//--------------------------------------------------------------------------------------
// Cyclic action
	IF (stStateMachine.intState=stStateMachine.intStateLastCycle) THEN
		// Simulation
		IF (SIf.stCfg.bolSimulation) THEN
			IF (((SIf.stMove.lreActPos+fbMcRelMove.Distance)<SIf.stMove.lreSWLimitPos_mm) AND (fbMcRelMove.Distance>0)AND (SIf.stMove.lreActPos<(lreActPos_old+fbMcRelMove.Distance))) THEN
				SIf.stMove.lreActPos := SIf.stMove.lreActPos + (fbMcRelMove.Velocity*udiSimPosTime_ms)/1000;
				SIf.stMove.lreActVel := fbMcRelMove.Velocity;
				SIf.stStatus.bolInPos := FALSE;
			ELSIF (((SIf.stMove.lreActPos+fbMcRelMove.Distance)>SIf.stMove.lreSWLimitNeg_mm) AND (fbMcRelMove.Distance<0)AND (SIf.stMove.lreActPos>(lreActPos_old+fbMcRelMove.Distance))) THEN
				SIf.stMove.lreActPos := SIf.stMove.lreActPos - (fbMcRelMove.Velocity*udiSimPosTime_ms)/1000;
				SIf.stMove.lreActVel := fbMcRelMove.Velocity;
				SIf.stStatus.bolInPos := FALSE;
			ELSE
				SIf.stMove.lreSetSpeed := 0;
				SIf.stStatus.bolInPos := TRUE;
			END_IF
		END_IF

		// No change action
		//MC_MoveRelative starts a relative positioning procedure based on the current set position and monitors the axis movement over the whole travel path.
		fbMcRelMove.Velocity := SIf.stMove.lreSetSpeed;
		fbMcRelMove.Deceleration := SIf.stMove.lreSetDec;
		fbMcRelMove.Acceleration := SIf.stMove.lreSetAcc;
		fbMcRelMove.Jerk := SIf.stMove.lreSetJerk;
		fbMcRelMove.Distance := SIf.stMove.lreSetPos;
		fbMcRelMove.Execute := TRUE;
		
		// State Change Condition
		IF (fbMcRelMove.Error) AND (bolfpFirstCycleDone) THEN
			SIf.stErr.dwoErrorID := fbMcRelMove.ErrorID;
			stStateMachine.intStateNext := cPOD_STA_Error;
		ELSIF (SIf.intCmd=cPOD_CMD_STOP) THEN
			stStateMachine.intStateNext := cPOD_STA_StopBusy;
		ELSIF (SIf.intCmd<>cPOD_CMD_REL_MOVE) THEN
			stStateMachine.intStateNext := cPOD_STA_QStopBusy;
		ELSIF ((SIf.stCfg.bolSimulation AND SIf.stStatus.bolInPos) OR (fbMcRelMove.Done))  AND (bolfpFirstCycleDone) THEN
			IF (SIf.intCmd=cPOD_CMD_REL_MOVE) THEN
				SIf.intCmd := cPOD_CMD_DONE;
			END_IF;
			stStateMachine.intStateNext := cPOD_STA_WaitForJob;
		END_IF
		bolfpFirstCycleDone := TRUE; //at least one call at the end of the FUB needed!
	END_IF

//--------------------------------------------------------------------------------------
// Exit action
	IF (stStateMachine.intState<>stStateMachine.intStateNext) THEN
		fbMcRelMove.Execute := FALSE;
		IF (SIf.stCfg.bolSimulation) THEN
			SIf.stMove.lreActVel := 0;
		END_IF
	END_IF
END_METHOD

{attribute 'object_name' := 'sta_StopBusy'}
METHOD PROTECTED sta_StopBusy : BOOL
// state implemetation
//--------------------------------------------------------------------------------------
// Entry action
	IF (stStateMachine.intState<>stStateMachine.intStateLastCycle) THEN
		stStateMachine.intStateLastCycle := stStateMachine.intState;
		
		bolfpFirstCycleDone := FALSE;
		
		IF (SIf.stCfg.bolSimulation) THEN
			SIf.stMove.lreActVel := 0;
		END_IF
	END_IF


//--------------------------------------------------------------------------------------
// Cyclic action
	IF (stStateMachine.intState=stStateMachine.intStateLastCycle) THEN

		//MC_Stop stops an axis with a defined braking ramp and blocks the axis for any motion commands. This behavior qualifies the block for stops under special circumstances where the axis must be prevented from further motion.
		fbMcHalt.Deceleration := SIf.stMove.lreSetDec;
		fbMcHalt.Jerk := 0; //Jerk (≥0). If the value is 0, the jerk parameterised with the last Move command is used.
		fbMcHalt.Execute := TRUE;
	
		// State Change Condition
		IF (fbMcHalt.Error) THEN
			SIf.stErr.dwoErrorID := fbMcHalt.ErrorID;
			stStateMachine.intStateNext := cPOD_STA_Error;
		ELSIF (fbMcHalt.Done) OR (SIf.stCfg.bolSimulation) THEN
			IF (SIf.intCmd=cPOD_CMD_STOP) THEN
				SIf.intCmd := cPOD_CMD_DONE;
			END_IF;
			stStateMachine.intStateNext := cPOD_STA_WaitForJob;
		ELSIF (SIf.intCmd=cPOD_CMD_CTRL_OFF) THEN
			stStateMachine.intStateNext := cPOD_STA_QStopBusy;
		END_IF
		bolfpFirstCycleDone := TRUE; //at least one call at the end of the FUB needed!
	END_IF




//--------------------------------------------------------------------------------------
// Exit action
	IF (stStateMachine.intState<>stStateMachine.intStateNext) THEN
		fbMcHalt.Execute := FALSE;
	END_IF
END_METHOD

{attribute 'object_name' := 'sta_WaitForJob'}
METHOD PROTECTED sta_WaitForJob : BOOL
// state implemetation
//--------------------------------------------------------------------------------------
// Entry action
	IF (stStateMachine.intState<>stStateMachine.intStateLastCycle) THEN
		stStateMachine.intStateLastCycle := stStateMachine.intState;
		
	END_IF


//--------------------------------------------------------------------------------------
// Cyclic action
	IF (stStateMachine.intState=stStateMachine.intStateLastCycle) THEN

		// State Change Condition
		IF (SIf.intCmd=cPOD_CMD_CTRL_OFF) THEN
			stStateMachine.intStateNext := cPOD_STA_PowerOff;
		ELSIF (SIf.intCmd=cPOD_CMD_CTRL_ON) THEN
			SIf.intCmd := cPOD_CMD_DONE;
		ELSIF (SIf.intCmd=cPOD_CMD_HOME) THEN
			stStateMachine.intStateNext := cPOD_STA_HomeBusy;
		ELSIF (SIf.intCmd=cPOD_CMD_REL_MOVE) THEN
			stStateMachine.intStateNext := cPOD_STA_RelMoveBusy;
		ELSIF (SIf.intCmd=cPOD_CMD_ABS_MOVE) THEN
			stStateMachine.intStateNext := cPOD_STA_AbsMoveBusy;
		ELSIF (SIf.intCmd=cPOD_CMD_MOD_MOVE) THEN
			stStateMachine.intStateNext := cPOD_STA_ModMoveBusy;
		ELSIF (SIf.intCmd=cPOD_CMD_POS_MOVE) THEN
			stStateMachine.intStateNext := cPOD_STA_PosMoveBusy;
		ELSIF (SIf.intCmd=cPOD_CMD_NEG_MOVE) THEN
			stStateMachine.intStateNext := cPOD_STA_NegMoveBusy;
		ELSIF (SIf.intCmd=cPOD_CMD_POS_JOG) THEN
			stStateMachine.intStateNext := cPOD_STA_PosJogBusy;
		ELSIF (SIf.intCmd=cPOD_CMD_NEG_JOG) THEN
			stStateMachine.intStateNext := cPOD_STA_NegJogBusy;
		ELSIF (SIf.intCmd=cPOD_CMD_STOP) THEN
			stStateMachine.intStateNext := cPOD_STA_StopBusy;
		ELSIF (SIf.intCmd=cPOD_CMD_EMCY_STOP_CTRL_OFF) THEN
			stStateMachine.intStateNext := cPOD_STA_QStopBusy;	
		END_IF
		
	END_IF


//--------------------------------------------------------------------------------------
// Exit action
	IF (stStateMachine.intState<>stStateMachine.intStateNext) THEN
		;
	END_IF
END_METHOD

{attribute 'object_name' := 'StateMachine'}
METHOD PROTECTED StateMachine : BOOL

// main statemachine of base controller
CASE stStateMachine.intState OF
	cPOD_STA_PowerOff: 
        THIS^.sta_PowerOff();
    cPOD_STA_PowerOnBusy: 
        THIS^.sta_PowerOnBusy();
	cPOD_STA_WaitForJob: 
        THIS^.sta_WaitForJob();
    cPOD_STA_HomeBusy: 
        THIS^.sta_HomeBusy();
	cPOD_STA_RelMoveBusy: 
        THIS^.sta_RelMoveBusy();
    cPOD_STA_AbsMoveBusy: 
        THIS^.sta_AbsMoveBusy();
	cPOD_STA_ModMoveBusy: 
        THIS^.sta_ModMoveBusy();
	cPOD_STA_PosMoveBusy: 
        THIS^.sta_PosMoveBusy();
	cPOD_STA_PosJogBusy: 
        THIS^.sta_PosJogBusy();
	cPOD_STA_NegMoveBusy: 
        THIS^.sta_NegMoveBusy();
	cPOD_STA_NegJogBusy: 
        THIS^.sta_NegJogBusy();
	cPOD_STA_QStopBusy: 
        THIS^.sta_QStopBusy();
	cPOD_STA_StopBusy: 
        THIS^.sta_StopBusy();
    cPOD_STA_Error: 
        THIS^.sta_Error();
END_CASE;
END_METHOD

{attribute 'object_name' := 'StateMachine_Service'}
METHOD PROTECTED StateMachine_Service : BOOL

IF (SIf.stCfg.bolSimulation) THEN
	SIf.stService.strValue := 'not available in simulation';
	SIf.intServiceCmd := cPOD_CMD_DONE;
ELSE

	// main statemachine of base controller
	CASE SIf.intServiceCmd OF
		cPOD_SCMD_WRITE_PARA: 
			THIS^.sJobWriteParameter();
		cPOD_SCMD_READ_PARA: 
			THIS^.sJobReadParameter();
		cPOD_SCMD_READ_PARA_NC: 
			THIS^.sJobReadParameterNC();
		cPOD_SCMD_WRITE_PARA_NC: 
			THIS^.sJobWriteParameterNC();
	ELSE
		SIf.intServiceCmd := POD_Cmd.cPOD_CMD_DONE;	
	END_CASE;
	
	// reset fb in same cycle as reset job -> done -> next job 
	IF (SIf.intServiceCmd = POD_Cmd.cPOD_CMD_DONE) THEN
		
		usiCaseScmd := 0;
		
		// reset FB calls - no cyclic calls!
		IF (fbEcCoeSdoWrite.bExecute) THEN
			fbEcCoeSdoWrite.bExecute := FALSE;
			fbEcCoeSdoWrite();
		END_IF
		IF (fbEcCoeSdoRead.bExecute) THEN
			fbEcCoeSdoRead.bExecute := FALSE;
			fbEcCoeSdoRead();
		END_IF
		IF (fbMCReadParameter.Enable) THEN
			fbMCReadParameter.Enable := FALSE;
			fbMCReadParameter(Axis := fbAxis);
		END_IF
		IF (fbMCReadBoolParameter.Enable) THEN
			fbMCReadBoolParameter.Enable := FALSE;
			fbMCReadBoolParameter(Axis := fbAxis);
		END_IF
		IF (fbMCWriteParameter.Execute) THEN
			fbMCWriteParameter.Execute := FALSE;
			fbMCWriteParameter(Axis := fbAxis);
		END_IF
		IF (fbMCWriteBoolParameter.Execute) THEN
			fbMCWriteBoolParameter.Execute := FALSE;
			fbMCWriteBoolParameter(Axis := fbAxis);
		END_IF
	END_IF
END_IF
END_METHOD

END_FUNCTION_BLOCK

// POUs/Controller/Driver/PTR [Paper Tracker]/FB_PTR
FUNCTION_BLOCK PUBLIC FB_PTR
VAR_INPUT
	In_uinBeltSpeed		: UINT;
END_VAR
VAR_OUTPUT
END_VAR
VAR
	m_udiTimeBase_us			: UDINT;		// Time base in [usec]
	m_intPaperOnBelt			: INT;			// # of Paper on the belt 
	m_intFirstPaperIdx			: INT;			// Index of the leading paper on the belt
	m_intLastPaperIdx			: INT;			// Index of the last paper on the belt
	m_arBuffer					: ARRAY[0..THIS^.cMAXBUFFERSIZE-1] OF T_PTR_STRUCT;
	m_arPositionList			: ARRAY[0..THIS^.cMAXBUFFERSIZE-1] OF T_PTR_STRUCT;
	m_intPaperEntryOffset_mm	: INT;
	m_dinBeltLength				: DINT;
	
	iIdx					: INT;
	iNdx					: INT;
	iDifference				: DINT;
END_VAR
VAR CONSTANT
	cMAXBUFFERSIZE					: INT  := 20;
	cPAPERPOSITION_TOLERANCE_mm		: UINT := 200;
END_VAR

IF m_intPaperOnBelt > 0 THEN
	iNdx := m_intFirstPaperIdx;
	
	FOR iIdx := 0 TO m_intPaperOnBelt-1 DO
		m_arBuffer[iNdx].udiTimeOnBelt_us := m_arBuffer[iNdx].udiTimeOnBelt_us + THIS^.m_udiTimeBase_us;
		m_arBuffer[iNdx].lrePositionOnBelt_mm := m_arBuffer[iNdx].lrePositionOnBelt_mm + UDINT_TO_LREAL(THIS^.m_udiTimeBase_us) * UDINT_TO_LREAL(THIS^.In_uinBeltSpeed) / 1000000.0;
				
		CASE m_arBuffer[iNdx].eStatus OF
			E_PTR_Status.EnterBusy:
				m_arBuffer[iNdx].lrePositionOnBeltAdjusted_mm := MIN(m_intPaperEntryOffset_mm, LREAL_TO_INT(m_arBuffer[iNdx].lrePositionOnBelt_mm));
				iDifference := m_intPaperEntryOffset_mm - LREAL_TO_DINT(m_arBuffer[iNdx].lrePositionOnBelt_mm);
					
				IF 	(iDifference < 0) AND (ABS(iDifference) > cPAPERPOSITION_TOLERANCE_mm) THEN
					m_arBuffer[iNdx].eStatus := E_PTR_Status.ERROR;
				END_IF
			E_PTR_Status.OnBelt:
				m_arBuffer[iNdx].lrePositionOnBeltAdjusted_mm := MIN(m_dinBeltLength, LREAL_TO_DINT(m_arBuffer[iNdx].lrePositionOnBelt_mm));
				iDifference := m_dinBeltLength - LREAL_TO_DINT(m_arBuffer[iNdx].lrePositionOnBelt_mm);

				IF 	(iDifference < 0) AND (ABS(iDifference) > cPAPERPOSITION_TOLERANCE_mm) THEN
					m_arBuffer[iNdx].eStatus :=  E_PTR_Status.ERROR;
				END_IF
			E_PTR_Status.ExitBusy:
		END_CASE
		
		m_arPositionList[iIdx] :=  m_arBuffer[iNdx];	
		iNdx := (iNdx + 1) MOD THIS^.cMAXBUFFERSIZE;
	END_FOR
ELSE
	m_arPositionList[0].eStatus := E_PTR_Status.Gone;
END_IF

PROPERTY PUBLIC BeltLength : DINT
GET
BeltLength := m_dinBeltLength;
END_GET
SET
m_dinBeltLength := BeltLength;
END_SET
END_PROPERTY

METHOD PUBLIC EnterComplete : BOOL
VAR_INPUT
END_VAR
m_arBuffer[m_intLastPaperIdx].eStatus := E_PTR_Status.OnBelt;
m_arBuffer[m_intLastPaperIdx].lrePositionOnBelt_mm := INT_TO_LREAL(m_intPaperEntryOffset_mm);
m_arBuffer[m_intLastPaperIdx].lrePositionOnBeltAdjusted_mm := INT_TO_LREAL(m_intPaperEntryOffset_mm);
END_METHOD

METHOD FB_init : BOOL
VAR_INPUT
	bInitRetains : BOOL; // if TRUE, the retain variables are initialized (warm start / cold start)
	bInCopyCode : BOOL;  // if TRUE, the instance afterwards gets moved into the copy code (online change)
END_VAR
m_udiTimeBase_us := 2000;
m_intPaperEntryOffset_mm := 0;
Reset();
END_METHOD

METHOD PUBLIC Insert : BOOL
VAR_INPUT
	uinPosition_mm			: UINT;
	udiItemId				: UDINT;
END_VAR
VAR
	iIdx					: INT;
	iNdx					: INT;
	iInsertIdx				: INT;
END_VAR
iInsertIdx := m_intFirstPaperIdx;
iNdx := m_intFirstPaperIdx;
iIdx := 0;
	
WHILE (iIdx < m_intPaperOnBelt) AND (uinPosition_mm < m_arBuffer[iNdx].lrePositionOnBelt_mm) DO
	iIdx := iIdx + 1;
	iNdx := (iNdx + 1) MOD THIS^.cMAXBUFFERSIZE;
END_WHILE
END_METHOD

PROPERTY PUBLIC PaperEntryOffset : INT
GET
PaperEntryOffset := m_intPaperEntryOffset_mm;
END_GET
SET
m_intPaperEntryOffset_mm := PaperEntryOffset;
END_SET
END_PROPERTY

PROPERTY PUBLIC PaperOnBelt : UINT
GET
PaperOnBelt := INT_TO_UINT(m_intPaperOnBelt);
END_GET
SET
END_SET
END_PROPERTY

METHOD PUBLIC Pop : T_PTR_STRUCT
// Remove a paper from the buffer
VAR_INPUT
END_VAR
Pop.eStatus := E_PTR_Status.Gone;
Pop.lrePositionOnBelt_mm := 0.0;
Pop.lrePositionOnBeltAdjusted_mm := 0.0;
Pop.udiItemId := 0;
Pop.udiTimeOnBelt_us := 0;


IF m_intPaperOnBelt > 0 THEN
	Pop := m_arBuffer[m_intFirstPaperIdx];
	m_arBuffer[m_intFirstPaperIdx].udiItemId := 0;
	m_arBuffer[m_intFirstPaperIdx].lrePositionOnBelt_mm := 0.0;
	m_arBuffer[m_intFirstPaperIdx].lrePositionOnBeltAdjusted_mm := 0.0;
	m_arBuffer[m_intFirstPaperIdx].udiTimeOnBelt_us := 0;
	m_arBuffer[m_intFirstPaperIdx].eStatus := E_PTR_Status.Gone;
	m_intPaperOnBelt := m_intPaperOnBelt - 1;

	IF m_intPaperOnBelt = 0 THEN
		m_arPositionList[0] := m_arBuffer[m_intFirstPaperIdx];
	END_IF

	m_intFirstPaperIdx := (m_intFirstPaperIdx + 1) MOD THIS^.cMAXBUFFERSIZE;
END_IF
END_METHOD

PROPERTY PUBLIC PositionList : POINTER TO T_PTR_STRUCT
GET
VAR
	iIdx			: INT;
	iNdx			: INT;
END_VAR
PositionList := ADR(m_arPositionList);
END_GET
SET
END_SET
END_PROPERTY

METHOD PUBLIC Push : BOOL
// Add (Push) a paper into the buffer
// Return an ID for the paper
VAR_INPUT
	In_udiItemId			: UDINT;
END_VAR
Push := FALSE;

IF m_intPaperOnBelt < THIS^.cMAXBUFFERSIZE THEN
	m_intLastPaperIdx := (m_intLastPaperIdx + 1) MOD THIS^.cMAXBUFFERSIZE;
	m_arBuffer[m_intLastPaperIdx].udiItemId := In_udiItemId;
	m_arBuffer[m_intLastPaperIdx].lrePositionOnBelt_mm := 0.0;
	m_arBuffer[m_intLastPaperIdx].lrePositionOnBeltAdjusted_mm := 0.0;
	m_arBuffer[m_intLastPaperIdx].udiTimeOnBelt_us := 0;
	m_arBuffer[m_intLastPaperIdx].eStatus := E_PTR_Status.EnterBusy;
	m_intPaperOnBelt := m_intPaperOnBelt + 1;
	Push := TRUE;
END_IF
END_METHOD

METHOD PUBLIC Reset : BOOL
VAR_INPUT
END_VAR
m_intFirstPaperIdx := 0;
m_intLastPaperIdx := -1;
m_intPaperOnBelt := 0;
END_METHOD

PROPERTY PUBLIC TimeBase : UDINT
GET
TimeBase := m_udiTimeBase_us;
END_GET
SET
m_udiTimeBase_us := TimeBase;
END_SET
END_PROPERTY

END_FUNCTION_BLOCK

// POUs/Controller/Driver/TCP (TCP communication driver)/FB_TCP
FUNCTION_BLOCK FB_TCP EXTENDS FB_CtrlBase
VAR
	/// Specific interface struct for public access
	SIf: T_Ctrl_SIf_TCP;
	intSendState: INT := 0;
	fbClientConnection: TC2_TCPIP.FB_ClientServerConnection;
	fbSend: TC2_TCPIP.FB_SocketSend;
	fbReceive: TC2_TCPIP.FB_SocketReceive;
	/// buffer for received messages
	fbReceiveBuffer: FB_DataSetFifo;
	/// buffer for messages to be sent
	fbSendBuffer: FB_DataSetFifo;
	stNextHead: ST_Header;
	bReceivedAck: BOOL;
	bReceivedNack: BOOL;
	iSendSize: UDINT;
	iNumSendTry: INT;
	tonSendTime: TON;
	pSendHeader: POINTER TO ST_Header;
	pByteSend: POINTER TO ARRAY[0..MAX_DATASET_SIZE] OF BYTE;
	pReceiveHead: POINTER TO ST_Header;
	pByteReceive: POINTER TO ARRAY[0..MAX_DATASET_SIZE] OF BYTE;
	naReceiveData: ARRAY[0..MAX_DATASET_SIZE] OF BYTE;
	pReceiveData: POINTER TO ARRAY[0..MAX_DATASET_SIZE] OF BYTE;
END_VAR
VAR CONSTANT
	cSendIdle: INT := 0;
	cSendBusy: INT := 1;
	cSendWait: INT := 2;
END_VAR

(*__________________________________________________________________________________________________
¦	
¦	Vistaprint Schweiz GmbH
¦	CH - 8401 Winterthur
¦
¦	www.vistaprint.ch - info@vistaprint.ch
¦___________________________________________________________________________________________________

Function desription:



History:
Version		Date			Author		Comment
---------------------------------------------------------------------------------------------------
0.00.1		21.05.2014		AVME/DSC	Start history. Based on TCP client from jetter prototyp (Sonja Segmueller)
___________________________________________________________________________________________________*)


SUPER^();

{attribute 'object_name' := 'Always'}
METHOD PROTECTED Always : BOOL
// not inherite from base !!!  special behaviour for this TCP driver
// SUPER^.Always();

// Conditions Always
IF (me.bolChangeBackToAUTO=TRUE) THEN // switch mode to automatic switch off controller
	//me.StateMachine.intStateNext := cSTA_OFFBusy;
	me.bolChangeBackToAUTO := FALSE;
END_IF

IF (CIf.SwCfg.bolExist=FALSE) THEN // hardware of controller does not exist
	me.StateMachine.intStateNext := cSTA_SINGLE_ANSWER;
ELSE
	;
END_IF

// ----------------------------------------------------------------------------------
// cyclic actions outside of statemachine
IF (me.StateMachine.intState<>cSTA_SINGLE_ANSWER) THEN
	
	// Cyclic call of the client connection
	fbClientConnection();	
END_IF
END_METHOD

{attribute 'object_name' := 'CtrlInit'}
METHOD CtrlInit : BOOL
// one time first cyclic call
// The socket is closed
SUPER^.CtrlInit();

me.StateMachine.intStateNext := TCP_CmdState.cSTA_Close;
END_METHOD

PROPERTY CtrlSIf : POINTER TO T_Ctrl_SIf_TCP
GET
CtrlSIf := ADR(SIf);
END_GET
END_PROPERTY

{attribute 'object_name' := 'CycleEndDuty'}
METHOD PROTECTED CycleEndDuty : BOOL
SUPER^.CycleEndDuty();

SendDataSequence();
END_METHOD

{attribute 'object_name' := 'CycleStartDuty'}
METHOD PROTECTED CycleStartDuty : BOOL
SUPER^.CycleStartDuty();

ReceiveDataSequence();
END_METHOD

{attribute 'object_name' := 'FB_init'}
METHOD FB_init : BOOL
VAR_INPUT
	/// if TRUE, the retain variables are initialized (warm start / cold start)
	bInitRetains: BOOL;
	/// if TRUE, the instance afterwards gets moved into the copy code (online change)
	bInCopyCode: BOOL;
END_VAR
VAR
	iIdx: UINT;
	iLength: UINT;
END_VAR
// ------------------------------------------------------------------------------------------------------------------------
// to manually change in new FUB implementation!!!
// define valid commands for this controller
iLength := SIZEOF(CIf.Job.aCmdList)/SIZEOF(CIf.Job.aCmdList[0]);
iIdx := 0;

WHILE (iIdx < iLength) AND (CIf.Job.aCmdList[iIdx].intCmd <> cCMD_INITIALIZED) DO
	iIdx := iIdx + 1; 
END_WHILE

IF (iIdx < iLength) THEN
// Add configuration of own comands	
	CIf.Job.aCmdList[iIdx].intCmd := TCP_CmdState.cCMD_Close;
	CIf.Job.aCmdList[iIdx].strName := 'CLOSE'; 
	CIf.Job.aCmdList[iIdx].bolAvailable := TRUE;
    iIdx := iIdx + 1;
		CIf.Job.aCmdList[iIdx].intCmd := TCP_CmdState.cCMD_Connect;
	CIf.Job.aCmdList[iIdx].strName := 'CONNECT'; 
	CIf.Job.aCmdList[iIdx].bolAvailable := TRUE;
    iIdx := iIdx + 1;

ELSE
	// Error if the aCmdList Array is to small
END_IF

// set name of class/typ
CIf.Info.strType := 'FB_TCP';
CIf.Info.strFullName := 'TCP Communication Driver';

// set alarm class
SIf.Alm[E_ALM_TCP.AddToReceiveBufferFailed].eAlmClass := E_AlmClass.INFO;
SIf.Alm[E_ALM_TCP.AddToReceiveBufferFailed].strText := 'addReceiveBufferFailed'; 
SIf.Alm[E_ALM_TCP.AddToSendBufferFailed].eAlmClass := E_AlmClass.INFO;
SIf.Alm[E_ALM_TCP.AddToSendBufferFailed].strText := 'addSendBufferFailed'; 
SIf.Alm[E_ALM_TCP.GetFromReceiveBufferFailed].eAlmClass := E_AlmClass.INFO;
SIf.Alm[E_ALM_TCP.GetFromReceiveBufferFailed].strText := 'getReceiveBufferFailed'; 
SIf.Alm[E_ALM_TCP.GetFromSendBufferFailed].eAlmClass := E_AlmClass.INFO;
SIf.Alm[E_ALM_TCP.GetFromSendBufferFailed].strText := 'getSendBufferFailed'; 
SIf.Alm[E_ALM_TCP.RemoveFromReceiveBufferFailed].eAlmClass := E_AlmClass.INFO;
SIf.Alm[E_ALM_TCP.RemoveFromReceiveBufferFailed].strText := 'RemoveReceiveBufferFailed'; 
SIf.Alm[E_ALM_TCP.RemoveFromSendBufferFailed].eAlmClass := E_AlmClass.INFO;
SIf.Alm[E_ALM_TCP.RemoveFromSendBufferFailed].strText := 'RemoveSendBufferFailed'; 
SIf.Alm[E_ALM_TCP.SocketConnectionLost].eAlmClass := E_AlmClass.INFO;
SIf.Alm[E_ALM_TCP.SocketConnectionLost].strText := 'SocketLost'; 
SIf.Alm[E_ALM_TCP.NotSent].eAlmClass := BASE_PLC.E_AlmClass.INFO;
SIf.Alm[E_ALM_TCP.NotSent].strText := 'NotSent';
SIf.Alm[E_ALM_TCP.NoAckReceived].eAlmClass := BASE_PLC.E_AlmClass.INFO;
SIf.Alm[E_ALM_TCP.NoAckReceived].strText := 'NoAckReceived';
SIf.Alm[E_ALM_TCP.FubErrorClientConnection].eAlmClass := BASE_PLC.E_AlmClass.INFO;
SIf.Alm[E_ALM_TCP.FubErrorClientConnection].strText := 'FUB error - client connection. Note add. info number';
SIf.Alm[E_ALM_TCP.FubErrorSendData].eAlmClass := BASE_PLC.E_AlmClass.INFO;
SIf.Alm[E_ALM_TCP.FubErrorSendData].strText := 'FUB error - send data. Note add. info number';
SIf.Alm[E_ALM_TCP.FubErrorReceiveData].eAlmClass := BASE_PLC.E_AlmClass.INFO;
SIf.Alm[E_ALM_TCP.FubErrorReceiveData].strText := 'FUB error - receive data. Note add. info number';


// *******************************************************************************
// initial values
// *******************************************************************************

// software configuration
CIf.SwCfg.bolExist := TRUE;
CIf.SwCfg.bolEnable := TRUE;
CIf.SwCfg.bolSimulation :=  FALSE;

// configuration
SIf.Cfg.bolAutoReconnectEnable  := TRUE;


// parameter
SIF.Par.strIPAdr := '192.168.2.182'; 
SIF.Par.udiPort := 7443;
SIF.Par.tTOConnection := T#10S;
SIF.Par.tTOReceive := T#5S;
SIF.Par.tTOSend := T#5S;
SIf.Par.iMaxWaitTimeAck := T#4S; // wait for Ack before declaring it not received
SIf.Par.iMaxSendTry := 5;

SIf.Cfg.bUsingAck := TRUE;

pReceiveData := ADR(naReceiveData);
pReceiveHead := pReceiveData;
END_METHOD

{attribute 'object_name' := 'getCmdState'}
METHOD PROTECTED getCmdState : STRING
VAR_INPUT
	intCmdState: INT;
	bolState: BOOL;
END_VAR
getCmdState := SUPER^.getCmdState(intCmdState:=intCmdState,bolState:=bolState); // get global/base defined cmds/states

IF (getCmdState='') THEN // global not defined get local
	// get string cmd/state string information in runtime	
	IF (bolState=FALSE) THEN
		// States's
		CASE intCmdState OF
			TCP_CmdState.cCMD_Connect: 
				getCmdState := 'cCMD_CONNECT';
			TCP_CmdState.cCMD_Close: 
				getCmdState := 'cCMD_CLOSE';

		END_CASE;
	ELSE
		// States's
		CASE intCmdState OF
			TCP_CmdState.cSTA_Close: 
				getCmdState := 'cSTA_CLOSE';
			TCP_CmdState.cSTA_CloseBusy: 
				getCmdState := 'cSTA_CLOSEBusy';
			TCP_CmdState.cSTA_Connect: 
				getCmdState := 'cSTA_CONNECT';
			TCP_CmdState.cSTA_ConnectBusy: 
				getCmdState := 'cSTA_CONNECTBusy';			
		END_CASE;
	END_IF 
END_IF
END_METHOD

{attribute 'object_name' := 'getCtrlSIf'}
METHOD getCtrlSIf : POINTER TO T_Ctrl_SIf_TCP
getCtrlSIf := ADR(SIf);
END_METHOD

{attribute 'object_name' := 'M_Pop'}
METHOD M_Pop : BOOL
VAR_OUTPUT
	naPopMsg: ARRAY[0..MAX_DATASET_SIZE] OF BYTE;
	bPop: BOOL;
END_VAR
IF fbReceiveBuffer.nCount > 0 THEN // there is something in the receive buffer
	fbReceiveBuffer.A_Remove( pHeader => pByteReceive );
	naPopMsg := pByteReceive^;
	M_Pop := 1;
	bPop := 1;
ELSE
	M_Pop := 0;
	bPop := 0;
END_IF
END_METHOD

{attribute 'object_name' := 'M_Push'}
METHOD M_Push : BOOL
VAR_INPUT
	paPushMsg: POINTER TO ARRAY[0..MAX_DATASET_SIZE] OF BYTE;
END_VAR
VAR
	pstPushMsg: POINTER TO ST_Header;
END_VAR
// send if desired
pstPushMsg := paPushMsg;
	
fbSendBuffer.A_Add(in := paPushMsg, iAddSize := UDINT_TO_INT(pstPushMsg^.udiMsgSize + SIZEOF(ST_HEADER)) , bOk=>M_Push );

IF NOT ( M_Push ) THEN 
	pfbAlarmCtrl^.setAlarm(CIf.Info.intCtrlId,E_ALM_TCP.AddToSendBufferFailed,0,ADR(SIf.Alm),E_AlmState.RST,CIf.Job.eMe_ActivAlmClass);
	me.StateMachine.intStateNext := BASE_PLC.cSTA_ERROR;
END_IF
END_METHOD

{attribute 'object_name' := 'ReceiveDataSequence'}
METHOD PROTECTED ReceiveDataSequence : BOOL
VAR
	bSuccess: BOOL;
	nLoad: UDINT;
	stACK: ST_Header;
END_VAR
// receive data if connected
IF (fbClientConnection.eState = TC2_TCPIP.E_SocketConnectionState.eSOCKET_CONNECTED) THEN
	IF fbReceive.bBusy THEN	
		fbReceive.bExecute := FALSE;
		fbReceive.sSrvNetId := '';
		fbReceive();
		
		IF NOT (fbReceive.bBusy) THEN
			// Receive is finished => see what we got
				
			// First Check about FUB error	
			IF (fbReceive.bError = TRUE) THEN
				IF NOT (SIf.Cur.bolFubErrorActive) THEN
					SIf.Cur.bolFubErrorActive:= TRUE;																				
					pfbAlarmCtrl^.setAlarm(CIf.Info.intCtrlId,E_ALM_TCP.FubErrorReceiveData, UDINT_TO_DINT(fbReceive.nErrId),ADR(SIf.Alm),E_AlmState.RST,CIf.Job.eMe_ActivAlmClass);																						
					// Try to close the socket. Needs reconnect for socket after an error!	
					me.StateMachine.intStateNext := TCP_CmdState.cSTA_CloseBusy;					
				END_IF	
				
			// No error			
			ELSE
				// Check received data
				CASE pReceiveHead^.uinMsgId  OF
					// ACK
					// **************************
					999: 
						bReceivedAck := 1;
					
					// NACK
					// **************************
					998: 
						bReceivedNack := 1;
						
					// Valid message IDs
					// **************************
					2, 3, 4, 5, 6, 7: 
					
						fbReceiveBuffer.A_Add(in := ADR(naReceiveData), iAddSize:= UDINT_TO_INT(SIZEOF(ST_Header) + pReceiveHead^.udiMsgSize), bOk=>bSuccess , nLoad => nLoad );
						IF NOT ( bSuccess ) THEN 
							pfbAlarmCtrl^.setAlarm(CIf.Info.intCtrlId,E_ALM_TCP.AddToReceiveBufferFailed,0,ADR(SIf.Alm),E_AlmState.RST,CIf.Job.eMe_ActivAlmClass);
							me.StateMachine.intStateNext := BASE_PLC.cSTA_ERROR;
							me.StateMachine.intState := BASE_PLC.cSTA_ERROR;
						END_IF
								
					// nothing has been received	
					// **************************
					0: 
					
				ELSE
					// send NACK Command
					IF(SIf.Cfg.bUsingAck) THEN
						stACK.uinMsgId := 998;
						fbSendBuffer.A_Add(in := ADR(stACK), bOk=>bSuccess , nLoad => nLoad, iAddSize:= SIZEOF(stACK.uinMsgId) );
						IF NOT (bSuccess) THEN 
							pfbAlarmCtrl^.setAlarm(CIf.Info.intCtrlId,E_ALM_TCP.AddToSendBufferFailed,0,ADR(SIf.Alm),E_AlmState.RST,CIf.Job.eMe_ActivAlmClass);
							me.StateMachine.intStateNext := BASE_PLC.cSTA_ERROR;
							me.StateMachine.intState := BASE_PLC.cSTA_ERROR;
						END_IF
					END_IF
				
				END_CASE
				// empty the receive data
				pReceiveHead^.uinMsgId := 0;			
			END_IF	
			
		END_IF
		
	// Trigger the next data receive 
	ELSE
		fbReceive(bExecute := FALSE); // Needs new trigger!
		fbReceive.sSrvNetId := '';
		fbReceive.hSocket := fbClientConnection.hSocket;
		fbReceive.cbLen := SIZEOF(naReceiveData);
		fbReceive.pDest := ADR(naReceiveData);
		fbReceive.tTimeout := SIf.Par.tTOReceive;
		fbReceive.bExecute := TRUE;
		fbReceive();
	END_IF
END_IF 
fbReceive();
END_METHOD

{attribute 'object_name' := 'SendDataSequence'}
METHOD PROTECTED SendDataSequence : BOOL
VAR
	intI: INT;
END_VAR
// Handle Send Data
CASE intSendState OF
	cSendIdle: 
		IF fbSendBuffer.nCount > 0 AND NOT (fbSend.bBusy) AND (fbClientConnection.eState = TC2_TCPIP.E_SocketConnectionState.eSOCKET_CONNECTED) THEN // there is something in the buffer that needs to be sent
			intSendState := cSendBusy;
			
			// Remove data from buffer. Get next package.
			fbSendBuffer.A_Get(pHeader => pSendHeader);
			pByteSend := pSendHeader;
			stNextHead := pSendHeader^;
			
			IF (stNextHead.uinMsgId = 999) OR (stNextHead.uinMsgId = 998 ) THEN // ack or nack
				iSendSize := SIZEOF(stNextHead.uinMsgId);
			ELSE
				iSendSize := stNextHead.udiMsgSize + SIZEOF(ST_Header);
			END_IF
			
			// send Command
			fbSend(bExecute := FALSE, sSrvNetId := ''); 
			fbSend.sSrvNetId := ''; // SIf.Par.strIPAdr;
			fbSend.hSocket := fbClientConnection.hSocket;
			fbSend.cbLen := iSendSize;
			fbSend.pSrc := pByteSend;
			fbSend.bExecute := TRUE;
			fbSend.tTimeout := SIf.Par.tTOSend;
			fbSend(); 
		ELSE
			fbSend.bExecute := FALSE;
			fbSend.sSrvNetId := '';
			fbSend();
		END_IF	
		// *)
	cSendBusy:
		IF NOT (fbSend.bBusy) THEN // sending done
			
			// First Check about FUB error	
			IF (fbSend.bError = TRUE) THEN
				IF NOT (SIf.Cur.bolFubErrorActive) THEN
					SIf.Cur.bolFubErrorActive:= TRUE;																				
					pfbAlarmCtrl^.setAlarm(CIf.Info.intCtrlId,E_ALM_TCP.FubErrorSendData, UDINT_TO_DINT(fbSend.nErrId),ADR(SIf.Alm),E_AlmState.RST,CIf.Job.eMe_ActivAlmClass);																						
					// Try to close the socket. Needs reconnect for socket after an error!	
					me.StateMachine.intStateNext := TCP_CmdState.cSTA_CloseBusy;					
				END_IF	
			// no error			
			ELSE
				IF (stNextHead.uinMsgId > 997) OR (NOT (SIf.Cfg.bUsingAck)) THEN // the sent was ack or nack
					fbSendBuffer.A_Remove();
					intSendState := cSendIdle;
				ELSE // wair for ack
					intSendState := cSendWait;
					tonSendTime(IN := 0);
					tonSendTime.PT := SIf.Par.iMaxWaitTimeAck;
					tonSendTime(IN := 1);
				END_IF	
			END_IF
			
		END_IF
		
		fbSend.bExecute := FALSE;
		fbSend.sSrvNetId := '';
		fbSend(); // *)
		
	cSendWait:
		fbSend.bExecute := FALSE;
		fbSend.sSrvNetId := '';
		fbSend();
		tonSendTime(IN := 1);
		// Wait for the ACK
		IF bReceivedAck THEN
			fbSendBuffer.A_Remove();
			bReceivedAck := 0;
			iNumSendTry := 0; // reset for next send
			intSendState := cSendIdle;
			
		ELSIF (tonSendTime.Q) OR (bReceivedNack) THEN // timeout
			
			iNumSendTry := iNumSendTry +1;
			IF iNumSendTry >= SIf.Par.iMaxSendTry THEN
				// the signal has not been acknoledged too many times => error
				pfbAlarmCtrl^.setAlarm(CIf.Info.intCtrlId,E_ALM_TCP.NoAckReceived,0,ADR(SIf.Alm),E_AlmState.RST,CIf.Job.eMe_ActivAlmClass);
				me.StateMachine.intStateNext := BASE_PLC.cSTA_ERROR;
			ELSE // retry sending
				fbSend.bExecute := TRUE;
				fbSend(); 
				intSendState := cSendBusy;
			END_IF
			
		END_IF
END_CASE // *)
fbSend();
END_METHOD

{attribute 'object_name' := 'sta_CLOSE'}
METHOD sta_CLOSE : BOOL
// state implemetation
// --------------------------------------------------------------------------------------
// Entry action
	IF (me.StateMachine.intState<>me.StateMachine.intStateLastCycle) THEN
		me.StateMachine.intStateLastCycle := me.StateMachine.intState;
		;
		
	END_IF

// --------------------------------------------------------------------------------------
// Cyclic action
	IF (me.StateMachine.intState=me.StateMachine.intStateLastCycle) THEN
		CASE me.intCmd OF
			TCP_CmdState.cCMD_Connect:
				me.StateMachine.intStateNext := TCP_CmdState.cSTA_ConnectBusy;
		END_CASE
	END_IF

// --------------------------------------------------------------------------------------
// Exit action
	IF (me.StateMachine.intState<>me.StateMachine.intStateNext) THEN
		;
	END_IF
END_METHOD

{attribute 'object_name' := 'sta_CLOSEBusy'}
METHOD sta_CLOSEBusy : BOOL
// state implemetation
// --------------------------------------------------------------------------------------
// Entry action
	IF (me.StateMachine.intState<>me.StateMachine.intStateLastCycle) THEN
		me.StateMachine.intStateLastCycle := me.StateMachine.intState;
		
		// Reset Tx state
		intSendState:= cSendIdle;
		fbSend.bExecute:= FALSE;
		fbReceive.bExecute:= FALSE;
		iNumSendTry := 0;
		
		// Close socket
		fbClientConnection.bEnable:= FALSE;
		
		IF me.intCmd = TCP_CmdState.cCMD_Close THEN
			// clear both buffers
			fbSendBuffer.A_Reset();
			fbReceiveBuffer.A_Reset();
		END_IF
	END_IF

// --------------------------------------------------------------------------------------
// Cyclic action
	IF (me.StateMachine.intState=me.StateMachine.intStateLastCycle) THEN
		
		// Check about FUB error	
		IF (fbClientConnection.bError = TRUE) OR (fbClientConnection.nErrId <> 0) THEN
			SIf.Cur.bolFubErrorActive:= TRUE;																					
			pfbAlarmCtrl^.setAlarm(CIf.Info.intCtrlId,E_ALM_TCP.FubErrorClientConnection, UDINT_TO_DINT(fbClientConnection.nErrId),ADR(SIf.Alm),E_AlmState.RST,CIf.Job.eMe_ActivAlmClass);																			
			me.StateMachine.intStateNext := BASE_PLC.cSTA_ERROR;	
		END_IF
					
		// Wait until socket is closed	
		IF (fbClientConnection.eState = TC2_TCPIP.E_SocketConnectionState.eSOCKET_DISCONNECTED) THEN 	
			IF me.intCmd = TCP_CmdState.cCMD_Close THEN
				me.StateMachine.intStateNext := TCP_CmdState.cSTA_Close;
			ELSE
				me.StateMachine.intStateNext := TCP_CmdState.cSTA_ConnectBusy;
			END_IF

		ELSIF (SIf.Cur.bolFubErrorActive) THEN
			me.StateMachine.intStateNext := BASE_PLC.cSTA_ERROR;	
		END_IF
		
	END_IF
	
// --------------------------------------------------------------------------------------
// Exit action
	IF (me.StateMachine.intState<>me.StateMachine.intStateNext) THEN
		;
	END_IF
END_METHOD

{attribute 'object_name' := 'sta_CONNECT'}
METHOD sta_CONNECT : BOOL
// state implemetation
// --------------------------------------------------------------------------------------
// Entry action
	IF (me.StateMachine.intState<>me.StateMachine.intStateLastCycle) THEN
		me.StateMachine.intStateLastCycle := me.StateMachine.intState;

		pfbAlarmCtrl^.setAlarm(CIf.Info.intCtrlId,E_ALM_TCP.SocketConnectionLost,0,ADR(SIf.Alm),E_AlmState.CLR,CIf.Job.eMe_ActivAlmClass);
	END_IF

// --------------------------------------------------------------------------------------
// Cyclic action
	IF (me.StateMachine.intState=me.StateMachine.intStateLastCycle) THEN
		// check if connection has been lost
		IF (fbClientConnection.eState <> TC2_TCPIP.E_SocketConnectionState.eSOCKET_CONNECTED) THEN 
			pfbAlarmCtrl^.setAlarm(CIf.Info.intCtrlId,E_ALM_TCP.SocketConnectionLost,0,ADR(SIf.Alm),E_AlmState.RST,CIf.Job.eMe_ActivAlmClass);
			
			IF SIf.Cfg.bolAutoReconnectEnable THEN
				me.StateMachine.intStateNext := TCP_CmdState.cSTA_CloseBusy;
			ELSE	
				me.StateMachine.intStateNext := BASE_PLC.cSTA_ERROR;
			END_IF
		END_IF
		
		CASE me.intCmd OF
			TCP_CmdState.cCMD_Close:
				me.StateMachine.intStateNext := TCP_CmdState.cSTA_CloseBusy;
			TCP_CmdState.cCMD_Connect:
				me.StateMachine.intStateNext := TCP_CmdState.cSTA_CloseBusy;
		END_CASE
	END_IF

// --------------------------------------------------------------------------------------
// Exit action
	IF (me.StateMachine.intState<>me.StateMachine.intStateNext) THEN
		;
	END_IF
END_METHOD

{attribute 'object_name' := 'sta_CONNECTBusy'}
METHOD sta_CONNECTBusy : BOOL
// state implemetation
// --------------------------------------------------------------------------------------
// Entry action
	IF (me.StateMachine.intState<>me.StateMachine.intStateLastCycle) THEN
		me.StateMachine.intStateLastCycle := me.StateMachine.intState;
		
		// Initialize and connect socket
		fbClientConnection.nMode := 0; 	// not used
		fbClientConnection.sRemoteHost := SIf.Par.strIPAdr;
		fbClientConnection.nRemotePort := SIf.Par.udiPort;
		fbClientConnection.tReconnect := SIF.Par.tTOConnection;
		fbClientConnection.bEnable:= TRUE;
	
		// clear both buffers
		fbSendBuffer.A_Reset();
		fbReceiveBuffer.A_Reset();
		
		// reset all nessecary parameters
		bReceivedAck := 0;
		bReceivedNack := 0;
		intSendState := 0;
	END_IF


// --------------------------------------------------------------------------------------
// Cyclic action
	IF (me.StateMachine.intState=me.StateMachine.intStateLastCycle) THEN
		
		// Check about FUB error	
		IF (fbClientConnection.bError = TRUE) OR (fbClientConnection.nErrId <> 0) THEN		
			SIf.Cur.bolFubErrorActive:= TRUE;																			
			pfbAlarmCtrl^.setAlarm(CIf.Info.intCtrlId,E_ALM_TCP.FubErrorClientConnection, UDINT_TO_DINT(fbClientConnection.nErrId),ADR(SIf.Alm),E_AlmState.RST,CIf.Job.eMe_ActivAlmClass);																			
			me.StateMachine.intStateNext := BASE_PLC.cSTA_ERROR;	
		END_IF
				
		// Wait for socket handle ID and connection state
		IF (fbClientConnection.hSocket.handle <> 0) AND (fbClientConnection.eState = TC2_TCPIP.E_SocketConnectionState.eSOCKET_CONNECTED) THEN 	
			me.StateMachine.intStateNext := TCP_CmdState.cSTA_Connect;
		END_IF
		
	END_IF

// --------------------------------------------------------------------------------------
// Exit action
	IF (me.StateMachine.intState<>me.StateMachine.intStateNext) THEN
		;
	END_IF
END_METHOD

{attribute 'object_name' := 'sta_ERROR'}
METHOD PROTECTED sta_ERROR : BOOL
// state implemetation
// --------------------------------------------------------------------------------------
// Entry action
	IF (me.StateMachine.intState<>me.StateMachine.intStateLastCycle) THEN
		me.StateMachine.intStateHistory := me.StateMachine.intStateLastCycle; // -> possibillity to go back to state before error
		me.StateMachine.intStateLastCycle := me.StateMachine.intState;
		
		// Clear pending commands
		CIf.Job.intACmd:= Base_PLC.cCMD_DONE;
		CIf.Job.intMCmd:= Base_PLC.cCMD_DONE;
			
		iNumSendTry := 0;
				
		// clear both buffers
		fbSendBuffer.A_Reset();
		fbReceiveBuffer.A_Reset();
		// Reset Tx state
		intSendState:= cSendIdle;
	END_IF
	

// --------------------------------------------------------------------------------------
// Cyclic action
	IF (me.StateMachine.intState=me.StateMachine.intStateLastCycle) THEN
		
		// State Change Condition
		IF (CIf.Job.bolAlmReset = TRUE) THEN
			SIf.Cur.bolFubErrorActive:= FALSE;
			me.StateMachine.intStateNext := cSTA_ERRORQuit;
		END_IF
	END_IF

// --------------------------------------------------------------------------------------
// Exit action
	IF (me.StateMachine.intState<>me.StateMachine.intStateNext) THEN
		;
	END_IF
END_METHOD

{attribute 'object_name' := 'sta_ERRORQuit'}
METHOD PROTECTED sta_ERRORQuit : BOOL
// state implemetation
// --------------------------------------------------------------------------------------
// Entry action
	IF (me.StateMachine.intState<>me.StateMachine.intStateLastCycle) THEN
		me.StateMachine.intStateLastCycle := me.StateMachine.intState;
		;
	END_IF

// -------------------------------------------------------------------------------------
// Cyclic action
	IF (me.StateMachine.intState=me.StateMachine.intStateLastCycle) THEN
		
		IF (CIf.Job.bolAlmReset = TRUE) THEN
			CIf.Job.eMe_ActivAlmClass := E_AlmClass.NONE; // reset feedback channel for parent
			CIf.Job.bolAlmReset := FALSE;
		END_IF
		
		// State Change Condition
		IF (CIf.Job.bolAlmReset = FALSE) THEN
			// Needs reconnect for socket after an error!	
			me.StateMachine.intStateNext := TCP_CmdState.cSTA_CloseBusy;
		END_IF
	END_IF

// --------------------------------------------------------------------------------------
// Exit action
	IF (me.StateMachine.intState<>me.StateMachine.intStateNext) THEN
		;
	END_IF
END_METHOD

{attribute 'object_name' := 'StateMachine'}
METHOD PROTECTED StateMachine : BOOL
SUPER^.StateMachine();

// main statemachine of base controller
CASE me.StateMachine.intState OF
	TCP_CmdState.cSTA_Close:
		THIS^.sta_CLOSE();
    TCP_CmdState.cSTA_ConnectBusy:
		THIS^.sta_CONNECTBusy();
	TCP_CmdState.cSTA_Connect:
		THIS^.sta_CONNECT();
	TCP_CmdState.cSTA_CloseBusy:
		THIS^.sta_CLOSEBusy();
END_CASE;
END_METHOD

END_FUNCTION_BLOCK

// POUs/Controller/Utility/FiFo/FB_DataSetFifo
FUNCTION_BLOCK FB_DataSetFifo
VAR_INPUT
	bOverwrite: BOOL;
	in: POINTER TO BYTE;
	iAddSize: INT;
END_VAR
VAR_OUTPUT
	bOk: BOOL;
	nCount: UDINT;
	nLoad: UDINT;
	out: ARRAY[0..MAX_DATASET_SIZE] OF BYTE;
	pHeader: POINTER TO ST_Header;
END_VAR
VAR
	/// Buffer memory used by FB_MemRingBuffer function block 
	arrBuffer: ARRAY[0..MAX_BUFFER_SIZE] OF BYTE;
	fbBuffer: FB_MemRingBuffer;
	intLoopRemove: INT;
	intLoopReset: INT;
END_VAR
VAR CONSTANT
	MAX_BUFFER_SIZE: UDINT := 1000;
END_VAR

;

ACTION A_Add:
fbBuffer.A_AddTail( pWrite:= in,
					cbWrite:= INT_TO_UDINT(iAddSize),
					pBuffer:= ADR( arrBuffer ),
					cbBuffer:= SIZEOF( arrBuffer ),
					bOk=> bOk,
					nCount => nCount );

IF NOT bOk THEN (* overflow ? *)
	IF bOverwrite THEN
		fbBuffer.A_RemoveHead(); (* remove one oldest entry *)
		fbBuffer.A_AddTail( bOk => bOk, nCount => nCount );
	END_IF
END_IF

nLoad := (fbBuffer.cbSize * 100) / MAX_BUFFER_SIZE;
END_ACTION

ACTION A_Get:
fbBuffer.A_GetHead( pRead:= ADR( out ),
					cbRead:= SIZEOF( out ),
					pBuffer:= ADR( arrBuffer ),
					cbBuffer:= SIZEOF( arrBuffer ),
					bOk=> bOk,
					nCount => nCount );

pHeader := ADR(out);					
					
nLoad := (fbBuffer.cbSize * 100) / MAX_BUFFER_SIZE;
END_ACTION

ACTION A_Remove:
// Clean up package buffer
FOR intLoopRemove:=0 TO SIZEOF(out)-1 DO
	out[intLoopRemove]:= 0;
END_FOR

// Remove data from buffer. Get next package.
fbBuffer.A_RemoveHead( 	pRead:= ADR(out),
						cbRead:= SIZEOF(out),
						pBuffer:= ADR(arrBuffer),
						cbBuffer:= SIZEOF(arrBuffer),
						bOk=> bOk,
						nCount => nCount );
// Return						
pHeader := ADR(out);

nLoad := (fbBuffer.cbSize * 100) / MAX_BUFFER_SIZE;
END_ACTION

ACTION A_Reset:
// MEMSET not working!
//MEMSET( ADR( arrBuffer ), 0, SIZEOF( arrBuffer ) ); (* reset (optional) internal buffer *)
FOR intLoopReset:=0 TO SIZEOF(arrBuffer)-1 DO
	arrBuffer[intLoopReset]:= 0;
END_FOR

fbBuffer.A_Reset( 	bOk=> bOk,
					nCount => nCount );

nLoad := (fbBuffer.cbSize * 100) / MAX_BUFFER_SIZE;
END_ACTION

END_FUNCTION_BLOCK

// POUs/Controller/Lvl0/GRR (Granulate Remote)/helper/cycle_Grr
FUNCTION cycle_Grr : BOOL
VAR_INPUT
	pGrr: POINTER TO T_GRR;
END_VAR

pGrr^.ctrl.fbGrr.In_bolAutoMode				:= pGrr^.io.In_bolAutoMode;
pGrr^.ctrl.fbGrr.In_bolEoffOrFuseOk			:= pGrr^.io.In_bolEoffOrFuseOk;
pGrr^.ctrl.fbGrr.In_bolMainPressureError	:= pGrr^.io.In_bolMainPressureError;
pGrr^.ctrl.fbGrr.In_bolPowderLowWarning		:= pGrr^.io.In_bolPowderLowWarning;
pGrr^.ctrl.fbGrr.In_bolSystemOk				:= pGrr^.io.In_bolSystemOk;
pGrr^.ctrl.fbGrr.In_intState				:= pGrr^.io.In_intState;
pGrr^.ctrl.fbGrr.In_bolToggleBitGrn			:= pGrr^.io.In_bolToggleBitGrn;
pGrr^.ctrl.fbGrr.In_intMainPressure			:= pGrr^.io.In_intMainPressure;
pGrr^.ctrl.fbGrr();
pGrr^.io.Out_intCommand						:= pGrr^.ctrl.fbGrr.Out_intCommand;
pGrr^.io.Out_intConveyorBelt				:= pGrr^.ctrl.fbGrr.Out_intConveyorBelt;
pGrr^.io.Out_intConveyorVibrator			:= pGrr^.ctrl.fbGrr.Out_intConveyorVibrator;
pGrr^.io.Out_intPowderVibrator				:= pGrr^.ctrl.fbGrr.Out_intPowderVibrator;
pGrr^.io.Out_uinFilterClearingCycleTime_min	:= pGrr^.ctrl.fbGrr.Out_uinFilterClearingCycleTime_min;
pGrr^.io.Out_bolToggleBitGrr				:= pGrr^.ctrl.fbGrr.Out_bolToggleBitGrr;
pGrr^.io.Out_intAnalogValue					:= pGrr^.ctrl.fbGrr.Out_intAnalogValue;

END_FUNCTION

// POUs/Controller/Lvl0/GRR (Granulate Remote)/helper/init_Grr
FUNCTION init_Grr : BOOL
VAR_INPUT
	pGrr			: POINTER TO T_GRR;
	/// instance array of all controller instances
	pCtrlInst		: POINTER TO fb_CtrlBase;
	/// common interface array of all controllers (main use for PLC)
	pCtrlCIf		: POINTER TO T_Ctrl_CIf;
END_VAR

pGrr^.ctrl.fbGrr.iniAllCtrlArrays(pCtrlInst,pCtrlCIf,pGrr^.id.Grr);

END_FUNCTION

// POUs/Controller/Lvl0/GRR (Granulate Remote)/FB_GRR
FUNCTION_BLOCK FB_GRR EXTENDS FB_CtrlBase
VAR_INPUT
	In_bolSystemOk: BOOL;
	In_bolMainPressureError: BOOL;
	In_bolEoffOrFuseOk: BOOL;
	In_bolPowderLowWarning: BOOL;
	In_bolAutoMode: BOOL;
	In_intState: INT;
	In_bolToggleBitGrn: BOOL;
	In_intMainPressure: INT;
END_VAR
VAR_OUTPUT
	Out_intCommand: INT;
	Out_intConveyorBelt: INT;
	Out_intPowderVibrator: INT;
	Out_intConveyorVibrator: INT;
	Out_uinFilterClearingCycleTime_min: UINT;
	Out_bolToggleBitGrr: BOOL;
	Out_intAnalogValue: INT;
END_VAR
VAR
	/// Specific interface struct for public access
	SIf: T_Ctrl_SIf_Grr;
	
	udiToggleBitGrrTimer_ms		: UDINT;
	udiToggleBitGrnTimer_ms		: UDINT;
	bToggleBitGrnOld			: BOOL;
	bToggleBitOK				: BOOL;
END_VAR

(*__________________________________________________________________________________________________
¦	
¦	Vistaprint Schweiz GmbH
¦	CH - 8401 Winterthur
¦
¦	www.vistaprint.ch - info@vistaprint.ch
¦___________________________________________________________________________________________________

Function desription:

History:
Version		Date			Author		Comment
---------------------------------------------------------------------------------------------------
0.00.1		05.11.2014		BB			Start history
0.00.2		06.02.2015		BB			changed name from GRN to GRR
___________________________________________________________________________________________________*)

SUPER^();

{attribute 'object_name' := 'Always'}
METHOD PROTECTED Always : BOOL
SUPER^.Always();

// ----------------------------------------------------------------------------------
// cyclic actions outside of statemachine
IF (me.StateMachine.intState <> cSTA_SINGLE_ANSWER) THEN
	
	// Toggle Bit Grr
	udiToggleBitGrrTimer_ms := udiToggleBitGrrTimer_ms + me.FUBInfo.udiSample_ms;
	IF (udiToggleBitGrrTimer_ms > 200) THEN
		SIf.Out.bolToggleBitGrr.intern := NOT SIf.Out.bolToggleBitGrr.intern;
		udiToggleBitGrrTimer_ms := 0;
	END_IF
	
	// check Toggle Bit Grn
	udiToggleBitGrnTimer_ms := udiToggleBitGrnTimer_ms + me.FUBInfo.udiSample_ms;
	IF (SIf.In.bolToggleBitGrn.intern <> bToggleBitGrnOld) THEN
		bToggleBitGrnOld := SIf.In.bolToggleBitGrn.intern;
		udiToggleBitGrnTimer_ms := 0;
	END_IF
	bToggleBitOK := FALSE;
	IF (udiToggleBitGrnTimer_ms < 1000) THEN
		bToggleBitOK := TRUE;
	END_IF
	
	IF NOT (bToggleBitOK) AND (me.StateMachine.intState <> cSTA_ERROR) AND (me.StateMachine.intState <> cSTA_ERRORQuit) THEN
		pfbAlarmCtrl^.setAlarm(CIf.Info.intCtrlId,E_ALM_GRR.LostConnection,0,ADR(SIf.Alm),E_AlmState.RST,CIf.Job.eMe_ActivAlmClass);
		me.StateMachine.intStateNext := Base_CmdState.cSTA_ERROR;
	END_IF
	
	IF NOT SIf.In.bolAutoMode.intern AND bToggleBitOK THEN
		IF (SIf.Cfg.bolManualModeAllowed) THEN
			pfbAlarmCtrl^.setAlarm(CIf.Info.intCtrlId,E_ALM_GRR.ManualModeWarning,0,ADR(SIf.Alm),E_AlmState.SET,CIf.Job.eMe_ActivAlmClass);
			pfbAlarmCtrl^.setAlarm(CIf.Info.intCtrlId,E_ALM_GRR.ManualModeError,0,ADR(SIf.Alm),E_AlmState.CLR,CIf.Job.eMe_ActivAlmClass);
		ELSIF (me.StateMachine.intState <> cSTA_ERROR) AND (me.StateMachine.intState <> cSTA_ERRORQuit) THEN
			pfbAlarmCtrl^.setAlarm(CIf.Info.intCtrlId,E_ALM_GRR.ManualModeError,0,ADR(SIf.Alm),E_AlmState.RST,CIf.Job.eMe_ActivAlmClass);
			pfbAlarmCtrl^.setAlarm(CIf.Info.intCtrlId,E_ALM_GRR.ManualModeWarning,0,ADR(SIf.Alm),E_AlmState.CLR,CIf.Job.eMe_ActivAlmClass);
			me.StateMachine.intStateNext := Base_CmdState.cSTA_ERROR;
		END_IF
	ELSE
		pfbAlarmCtrl^.setAlarm(CIf.Info.intCtrlId,E_ALM_GRR.ManualModeWarning,0,ADR(SIf.Alm),E_AlmState.CLR,CIf.Job.eMe_ActivAlmClass);
	END_IF
	
	IF SIf.In.bolPowderLowWarning.intern AND bToggleBitOK THEN
		pfbAlarmCtrl^.setAlarm(CIf.Info.intCtrlId,E_ALM_GRR.LowPowderWarning,0,ADR(SIf.Alm),E_AlmState.SET,CIf.Job.eMe_ActivAlmClass);
	ELSE
		pfbAlarmCtrl^.setAlarm(CIf.Info.intCtrlId,E_ALM_GRR.LowPowderWarning,0,ADR(SIf.Alm),E_AlmState.CLR,CIf.Job.eMe_ActivAlmClass);
	END_IF
	
	// reasons are either PressureError or SystemError (EOFF/Fuse/Motor)
	IF NOT SIf.In.bolSystemOk.intern AND bToggleBitOK THEN
		IF SIf.In.bolMainPressureError.intern THEN
			pfbAlarmCtrl^.setAlarm(CIf.Info.intCtrlId,E_ALM_GRR.PressureError,0,ADR(SIf.Alm),E_AlmState.RST,CIf.Job.eMe_ActivAlmClass);
			me.StateMachine.intStateNext := Base_CmdState.cSTA_OFFBusy;
		ELSE
			pfbAlarmCtrl^.setAlarm(CIf.Info.intCtrlId,E_ALM_GRR.SystemError,0,ADR(SIf.Alm),E_AlmState.RST,CIf.Job.eMe_ActivAlmClass);
			me.StateMachine.intStateNext := Base_CmdState.cSTA_OFFBusy;
		END_IF
	END_IF
	
	// Check Parameters
	// Conveyor Belt
	IF (SIf.Par.rConveyorBelt_Hz>SIf.Cfg.rMaxFreq_Hz) THEN
		SIf.Par.rConveyorBelt_Hz := SIf.Cfg.rMaxFreq_Hz;
	ELSIF (SIf.Par.rConveyorBelt_Hz<0) THEN
		SIf.Par.rConveyorBelt_Hz := 0;
	END_IF
	// Conveyor Vibrator
	IF (SIf.Par.rConveyorVibrator_Hz>SIf.Cfg.rMaxFreq_Hz) THEN
		SIf.Par.rConveyorVibrator_Hz := SIf.Cfg.rMaxFreq_Hz;
	ELSIF (SIf.Par.rConveyorVibrator_Hz<0) THEN
		SIf.Par.rConveyorVibrator_Hz := 0;
	END_IF
	// Powder Virbrator
	IF (SIf.Par.rPowderVibrator_Hz>SIf.Cfg.rMaxFreq_Hz) THEN
		SIf.Par.rPowderVibrator_Hz := SIf.Cfg.rMaxFreq_Hz;
	ELSIF (SIf.Par.rPowderVibrator_Hz<0) THEN
		SIf.Par.rPowderVibrator_Hz := 0;
	END_IF
	// Analog Value
	IF (SIf.Par.rAirKnife_p>100) THEN
		SIf.Par.rAirKnife_p := 100;
	ELSIF (SIf.Par.rAirKnife_p<0) THEN
		SIf.Par.rAirKnife_p := 0;
	END_IF
	
	// Set Outputs
	SIf.Out.intConveyorBelt.intern := REAL_TO_INT(MAX_INT/SIf.Cfg.rMaxFreq_Hz*SIf.Par.rConveyorBelt_Hz);
	SIf.Out.intConveyorVibrator.intern := REAL_TO_INT(MAX_INT/SIf.Cfg.rMaxFreq_Hz*SIf.Par.rConveyorVibrator_Hz);
	SIf.Out.intPowderVibrator.intern := REAL_TO_INT(MAX_INT/SIf.Cfg.rMaxFreq_Hz*SIf.Par.rPowderVibrator_Hz);
	SIf.Out.intAnalogValue.intern := REAL_TO_INT(MAX_INT/100*SIf.Par.rAirKnife_p);
	SIf.Out.uinFilterClearingCycleTime_min.intern := SIf.Par.uinFilterClearingCycleTime_min;
	
	// Set Current Values
	SIf.Cur.intMainPressure := SIf.In.intMainPressure.intern;

END_IF

// ----------------------------------------------------------------------------------
// overrule error always from base -> no EOFF State!! in EOFF go to OFF
IF (me.StateMachine.intStateNext = cSTA_EOFFBusy) THEN
	IF (me.StateMachine.intState = cSTA_OFF) THEN
		me.StateMachine.intStateNext := cSTA_OFF;
	ELSE // stay in OFF
		me.StateMachine.intStateNext := cSTA_OFFBusy;
	END_IF
END_IF
END_METHOD

PROPERTY PUBLIC CtrlSIf : POINTER TO T_Ctrl_SIf_GRR
GET
CtrlSIf := ADR(SIf);
END_GET
END_PROPERTY

{attribute 'object_name' := 'FB_init'}
METHOD FB_init : BOOL
VAR_INPUT
	/// if TRUE, the retain variables are initialized (warm start / cold start)
	bInitRetains: BOOL;
	/// if TRUE, the instance afterwards gets moved into the copy code (online change)
	bInCopyCode: BOOL;
END_VAR
VAR
	iIdx: UINT;
	iLength: UINT;
END_VAR
// ------------------------------------------------------------------------------------------------------------------------
// to manually change in new FUB implementation!!!
// define valid commands for this controller
iLength := SIZEOF(CIf.Job.aCmdList)/SIZEOF(CIf.Job.aCmdList[0]);
iIdx := 0;

WHILE (iIdx < iLength) AND (CIf.Job.aCmdList[iIdx].intCmd <> cCMD_INITIALIZED) DO
	iIdx := iIdx + 1; 
END_WHILE

IF (iIdx < iLength) THEN
	// Add configuration of own comands	
	CIf.Job.aCmdList[iIdx].intCmd := BASE_PLC.cCMD_RUN;
	CIf.Job.aCmdList[iIdx].strName := 'RUN'; 
	CIf.Job.aCmdList[iIdx].bolAvailable := TRUE;
    iIdx := iIdx + 1;
ELSE
	// Error if the aCmdList Array is to small
END_IF

// set name of class/typ
CIf.Info.strType := 'FB_GRR';
CIf.Info.strFullName := 'Granulate Remote';

// set alarm class
SIf.Alm[E_ALM_GRR.SystemError].eAlmClass := E_AlmClass.OFF;
SIf.Alm[E_ALM_GRR.SystemError].strText := 'System Error';
SIf.Alm[E_ALM_GRR.PressureError].eAlmClass := E_AlmClass.OFF;
SIf.Alm[E_ALM_GRR.PressureError].strText := 'Pressure Error';
SIf.Alm[E_ALM_GRR.LowPowderWarning].eAlmClass := E_AlmClass.WARNING;
SIf.Alm[E_ALM_GRR.LowPowderWarning].strText := 'Low Powder';
SIf.Alm[E_ALM_GRR.ManualModeWarning].eAlmClass := E_AlmClass.WARNING;
SIf.Alm[E_ALM_GRR.ManualModeWarning].strText := 'Manual Operation';
SIf.Alm[E_ALM_GRR.ManualModeError].eAlmClass := E_AlmClass.OFF;
SIf.Alm[E_ALM_GRR.ManualModeError].strText := 'Manual Operation';
SIf.Alm[E_ALM_GRR.LostConnection].eAlmClass := E_AlmClass.OFF;
SIf.Alm[E_ALM_GRR.LostConnection].strText := 'Lost Connection to the Granulate Machine';

// *******************************************************************************
// initial values
// *******************************************************************************

// software configuration
CIf.SwCfg.bolExist := TRUE;
CIf.SwCfg.bolEnable := TRUE;
CIf.SwCfg.bolSimulation := FALSE;

me.AlarmConfig.bolEOffAlarmTransitionDisable := TRUE;
me.AlarmConfig.bolOffAlarmTransitionDisable := TRUE;
me.AlarmConfig.bolEOffCmdTransitionDisable := TRUE;
me.AlarmConfig.bolOffCmdTransitionDisable := TRUE;

// configuration
SIf.Cfg.bolManualModeAllowed := FALSE;
SIf.Cfg.rMaxFreq_Hz := 50.0;

// parameter
SIf.Par.rConveyorBelt_Hz		:= SIf.Cfg.rMaxFreq_Hz/2;
SIf.Par.rConveyorVibrator_Hz	:= SIf.Cfg.rMaxFreq_Hz/2;
SIf.Par.rPowderVibrator_Hz		:= SIf.Cfg.rMaxFreq_Hz/2;
SIf.Par.rAirKnife_p				:= 50;
SIf.Par.uinFilterClearingCycleTime_min	:= 4*60;
END_METHOD

{attribute 'object_name' := 'getCmdState'}
METHOD PROTECTED getCmdState : STRING
VAR_INPUT
	intCmdState: INT;
	bolState: BOOL;
END_VAR
getCmdState := SUPER^.getCmdState(intCmdState:=intCmdState,bolState:=bolState); // get global/base defined cmds/states

IF (getCmdState='') THEN // global not defined get local
	// get string cmd/state string information in runtime	
	IF (bolState=FALSE) THEN
		// Commands
		;
	ELSE
		// States
		CASE intCmdState OF
			// Main states
			GRR_CmdState.cSTA_MANUALBusy:
				getCmdState := 'MANUALBusy';
			GRR_CmdState.cSTA_MANUAL:
				getCmdState := 'MANUAL';
		END_CASE;
	END_IF 
END_IF
END_METHOD

{attribute 'object_name' := 'IoInBridge'}
METHOD PROTECTED IoInBridge : BOOL
SUPER^.IoInBridge();
// digitale and analoge inputs read from hardware or forcing
SIf.In.bolSystemOk.map	:= THIS^.In_bolSystemOk;
SIf.In.bolMainPressureError.map	:= THIS^.In_bolMainPressureError;
SIf.In.bolEoffOrFuseOk.map	:= THIS^.In_bolEoffOrFuseOk;
SIf.In.bolPowderLowWarning.map	:= THIS^.In_bolPowderLowWarning;
SIf.In.bolAutoMode.map	:= THIS^.In_bolAutoMode;
SIf.In.intState.map	:= THIS^.In_intState;
SIf.In.bolToggleBitGrn.map	:= THIS^.In_bolToggleBitGrn;
SIf.In.intMainPressure.map	:= THIS^.In_intMainPressure;

IF (CIf.SwCfg.bolSimulation = FALSE) THEN
	BASE_PLC.getInBol(CIf.Job.bolIoForce,ADR(SIf.In.bolSystemOk));
	BASE_PLC.getInBol(CIf.Job.bolIoForce,ADR(SIf.In.bolMainPressureError));
	BASE_PLC.getInBol(CIf.Job.bolIoForce,ADR(SIf.In.bolEoffOrFuseOk));
	BASE_PLC.getInBol(CIf.Job.bolIoForce,ADR(SIf.In.bolPowderLowWarning));
	BASE_PLC.getInBol(CIf.Job.bolIoForce,ADR(SIf.In.bolAutoMode));
	BASE_PLC.getInInt(CIf.Job.bolIoForce,ADR(SIf.In.intState));
	BASE_PLC.getInBol(CIf.Job.bolIoForce,ADR(SIf.In.bolToggleBitGrn));
	BASE_PLC.getInInt(CIf.Job.bolIoForce,ADR(SIf.In.intMainPressure));
ELSE
	//simulation of global IO
	SIf.In.bolSystemOk.intern			:= TRUE;
	SIf.In.bolMainPressureError.intern	:= FALSE;
	SIf.In.bolEoffOrFuseOk.intern		:= TRUE;
	SIf.In.bolPowderLowWarning.intern	:= FALSE;
	SIf.In.bolAutoMode.intern			:= TRUE;
	SIf.In.intState.intern				:= SIf.Out.intCommand.intern;
	SIf.In.bolToggleBitGrn.intern		:= SIf.Out.bolToggleBitGrr.intern;
END_IF
END_METHOD

{attribute 'object_name' := 'IoOutBridge'}
METHOD PROTECTED IoOutBridge : BOOL
// digitale and analoge inputs read from hardware or forcing
IF (CIf.SwCfg.bolSimulation = FALSE) THEN
	setOutInt(CIf.Job.bolIoForce ,ADR(SIf.Out.intCommand));
	setOutInt(CIf.Job.bolIoForce ,ADR(SIf.Out.intConveyorBelt));
	setOutInt(CIf.Job.bolIoForce ,ADR(SIf.Out.intConveyorVibrator));
	setOutInt(CIf.Job.bolIoForce ,ADR(SIf.Out.intPowderVibrator));
	setOutUint(CIf.Job.bolIoForce ,ADR(SIf.Out.uinFilterClearingCycleTime_min));
	setOutBol(CIf.Job.bolIoForce ,ADR(SIf.Out.bolToggleBitGrr));
	setOutUint(CIf.Job.bolIoForce ,ADR(SIf.Out.intAnalogValue));
	
	THIS^.Out_intCommand := SIf.Out.intCommand.map;
	THIS^.Out_intConveyorBelt := SIf.Out.intConveyorBelt.map;
	THIS^.Out_intConveyorVibrator := SIf.Out.intConveyorVibrator.map;
	THIS^.Out_intPowderVibrator := SIf.Out.intPowderVibrator.map;
	THIS^.Out_uinFilterClearingCycleTime_min := SIf.Out.uinFilterClearingCycleTime_min.map;
	THIS^.Out_bolToggleBitGrr := SIf.Out.bolToggleBitGrr.map;
	THIS^.Out_intAnalogValue := SIf.Out.intAnalogValue.map;
ELSE
	THIS^.Out_intCommand := 0;
	THIS^.Out_intConveyorBelt := 0;
	THIS^.Out_intConveyorVibrator := 0;
	THIS^.Out_intPowderVibrator := 0;
	THIS^.Out_uinFilterClearingCycleTime_min := 0;
	THIS^.Out_bolToggleBitGrr := SIf.Out.bolToggleBitGrr.map;
	THIS^.Out_intAnalogValue := 0;
END_IF
END_METHOD

{attribute 'object_name' := 'sta_ERROR'}
METHOD PROTECTED sta_ERROR : BOOL
// state implemetation
// --------------------------------------------------------------------------------------
// Entry action
	IF (me.StateMachine.intState<>me.StateMachine.intStateLastCycle) THEN
		me.StateMachine.intStateHistory := me.StateMachine.intStateLastCycle; // -> possibillity to go back to state before error
		me.StateMachine.intStateLastCycle := me.StateMachine.intState;
	END_IF

	
// --------------------------------------------------------------------------------------
// Cyclic action
	
	// State Change Condition
	IF (CIf.Job.bolAlmReset = TRUE) THEN
		me.StateMachine.intStateNext := cSTA_ERRORQuit;
	END_IF

	
// --------------------------------------------------------------------------------------
// Exit action
	IF (me.StateMachine.intState<>me.StateMachine.intStateNext) THEN
		;
	END_IF
END_METHOD

{attribute 'object_name' := 'sta_ERRORQuit'}
METHOD PROTECTED sta_ERRORQuit : BOOL
// state implemetation
// --------------------------------------------------------------------------------------
// Entry action
	IF (me.StateMachine.intState<>me.StateMachine.intStateLastCycle) THEN
		me.StateMachine.intStateLastCycle := me.StateMachine.intState;
	END_IF

	
// --------------------------------------------------------------------------------------
// Cyclic action
	
	// evtl. wait time if reset of device is necessary and then decide to go to states or ERROR state
	IF (CIf.Job.bolAlmReset = TRUE) THEN
		CIf.Job.eMe_ActivAlmClass := E_AlmClass.NONE; // reset feedback channel for parent
		CIf.Job.bolAlmReset := FALSE;
	END_IF
	
	IF (SIf.In.bolAutoMode.intern) THEN
		me.StateMachine.intStateNext := Base_PLC.cSTA_OFFBusy;
	ELSE
		me.StateMachine.intStateNext := GRR_CmdState.cSTA_MANUALBusy;
	END_IF
	
// --------------------------------------------------------------------------------------
// Exit action
	IF (me.StateMachine.intState<>me.StateMachine.intStateNext) THEN
		;
	END_IF
END_METHOD

{attribute 'object_name' := 'sta_MANUAL'}
METHOD PROTECTED sta_MANUAL : BOOL
// state implemetation
// --------------------------------------------------------------------------------------
// Entry action
	IF (me.StateMachine.intState<>me.StateMachine.intStateLastCycle) THEN
		me.StateMachine.intStateLastCycle := me.StateMachine.intState;
	END_IF


// --------------------------------------------------------------------------------------
// Cyclic action

	IF (SIf.In.bolAutoMode.intern) THEN
		me.StateMachine.intStateNext := cSTA_OFFBusy;
	END_IF

	
// --------------------------------------------------------------------------------------
// Exit action
	IF (me.StateMachine.intState<>me.StateMachine.intStateNext) THEN
		;
	END_IF
END_METHOD

{attribute 'object_name' := 'sta_MANUALBusy'}
METHOD PROTECTED sta_MANUALBusy : BOOL
// state implemetation
// --------------------------------------------------------------------------------------
// Entry action
	IF (me.StateMachine.intState<>me.StateMachine.intStateLastCycle) THEN
		me.StateMachine.intStateLastCycle := me.StateMachine.intState;
		
		SIf.Out.intCommand.intern := cCMD_OFF;
	END_IF


// --------------------------------------------------------------------------------------
// Cyclic action

	IF (SIf.In.bolAutoMode.intern) THEN
		me.StateMachine.intStateNext := cSTA_OFFBusy;
	ELSE
		me.StateMachine.intStateNext := GRR_CmdState.cSTA_MANUAL;
	END_IF

	
// --------------------------------------------------------------------------------------
// Exit action
	IF (me.StateMachine.intState<>me.StateMachine.intStateNext) THEN
		;
	END_IF
END_METHOD

{attribute 'object_name' := 'sta_OFF'}
METHOD PROTECTED sta_OFF : BOOL
// state implemetation
// --------------------------------------------------------------------------------------
// Entry action
	IF (me.StateMachine.intState<>me.StateMachine.intStateLastCycle) THEN
		me.StateMachine.intStateLastCycle := me.StateMachine.intState;
	END_IF


// --------------------------------------------------------------------------------------
// Cyclic action

	IF (SIf.In.bolAutoMode.intern) THEN
		IF me.intCmd=Base_PLC.cCMD_RUN AND SIf.In.bolSystemOk.intern THEN
			me.StateMachine.intStateNext := Base_PLC.cSTA_RUNBusy;
		END_IF
	ELSE
		me.StateMachine.intStateNext := GRR_CmdState.cSTA_MANUALBusy;
	END_IF


// --------------------------------------------------------------------------------------
// Exit action
	IF (me.StateMachine.intState<>me.StateMachine.intStateNext) THEN
		;
	END_IF
END_METHOD

{attribute 'object_name' := 'sta_OFFBusy'}
METHOD PROTECTED sta_OFFBusy : BOOL
// state implemetation
// --------------------------------------------------------------------------------------
// Entry action
	IF (me.StateMachine.intState<>me.StateMachine.intStateLastCycle) THEN
		me.StateMachine.intStateLastCycle := me.StateMachine.intState;
		
		SIf.Out.intCommand.intern := cCMD_OFF;
	END_IF


// --------------------------------------------------------------------------------------
// Cyclic action

	IF (SIf.In.bolAutoMode.intern) THEN
		IF (SIf.In.intState.intern = cSTA_OFF) THEN
			me.StateMachine.intStateNext := cSTA_OFF;
		ELSIF me.intCmd=Base_PLC.cCMD_RUN AND SIf.In.bolSystemOk.intern THEN
			me.StateMachine.intStateNext := Base_PLC.cSTA_RUNBusy;
		END_IF
	ELSE
		me.StateMachine.intStateNext := GRR_CmdState.cSTA_MANUALBusy;
	END_IF

	
// --------------------------------------------------------------------------------------
// Exit action
	IF (me.StateMachine.intState<>me.StateMachine.intStateNext) THEN
		;
	END_IF
END_METHOD

{attribute 'object_name' := 'sta_PON'}
METHOD PROTECTED sta_PON : BOOL
// state implemetation
// --------------------------------------------------------------------------------------
// Entry action
	IF (me.StateMachine.intState<>me.StateMachine.intStateLastCycle) THEN
		me.StateMachine.intStateLastCycle := me.StateMachine.intState;
	END_IF

	
// --------------------------------------------------------------------------------------
// Cyclic action

	IF (SIf.In.bolAutoMode.intern) THEN
		IF (me.intCmd > Base_PLC.cCMD_PON) THEN
			me.StateMachine.intStateNext := Base_PLC.cSTA_OFFBusy;
		END_IF
	ELSE
		me.StateMachine.intStateNext := GRR_CmdState.cSTA_MANUALBusy;
	END_IF
	
	
// --------------------------------------------------------------------------------------
// Exit action
	IF (me.StateMachine.intState<>me.StateMachine.intStateNext) THEN
		;
	END_IF
END_METHOD

{attribute 'object_name' := 'sta_PONBusy'}
METHOD PROTECTED sta_PONBusy : BOOL
// state implemetation
// --------------------------------------------------------------------------------------
// Entry action
IF (me.StateMachine.intState<>me.StateMachine.intStateLastCycle) THEN
	me.StateMachine.intStateLastCycle := me.StateMachine.intState;
	
	IF (SIf.In.intState.intern < cSTA_PON) THEN
		SIf.Out.intCommand.intern := cCMD_PON;
	END_IF
END_IF


// --------------------------------------------------------------------------------------
// Cyclic action

	IF (SIf.In.intState.intern >= cSTA_PON) THEN
		me.StateMachine.intStateNext := cSTA_PON;
	END_IF


// --------------------------------------------------------------------------------------
// Exit action
IF (me.StateMachine.intState<>me.StateMachine.intStateNext) THEN
	;
END_IF
END_METHOD

{attribute 'object_name' := 'sta_RUN'}
METHOD PROTECTED sta_RUN : BOOL
// state implemetation
// --------------------------------------------------------------------------------------
// Entry action
	IF (me.StateMachine.intState<>me.StateMachine.intStateLastCycle) THEN
		me.StateMachine.intStateLastCycle := me.StateMachine.intState;
	END_IF


// --------------------------------------------------------------------------------------
// Cyclic action

	IF (SIf.In.bolAutoMode.intern) THEN
		IF me.intCmd=Base_PLC.cCMD_OFF THEN
			me.StateMachine.intStateNext := Base_PLC.cSTA_OFFBusy;
		END_IF
	ELSE
		me.StateMachine.intStateNext := GRR_CmdState.cSTA_MANUALBusy;
	END_IF


// --------------------------------------------------------------------------------------
// Exit action
	IF (me.StateMachine.intState<>me.StateMachine.intStateNext) THEN
		;
	END_IF
END_METHOD

{attribute 'object_name' := 'sta_RUNBusy'}
METHOD PROTECTED sta_RUNBusy : BOOL
// state implemetation
// --------------------------------------------------------------------------------------
// Entry action
	IF (me.StateMachine.intState<>me.StateMachine.intStateLastCycle) THEN
		me.StateMachine.intStateLastCycle := me.StateMachine.intState;
		
		SIf.Out.intCommand.intern := cCMD_RUN;
	END_IF


// --------------------------------------------------------------------------------------
// Cyclic action

	IF (SIf.In.bolAutoMode.intern) THEN
		IF me.intCmd=Base_PLC.cCMD_OFF THEN
			me.StateMachine.intStateNext := Base_PLC.cSTA_OFFBusy;
		ELSIF (SIf.In.intState.intern = cSTA_RUN) THEN
			me.StateMachine.intStateNext := Base_PLC.cSTA_RUN;
		END_IF
	ELSE
		me.StateMachine.intStateNext := GRR_CmdState.cSTA_MANUALBusy;
	END_IF


// --------------------------------------------------------------------------------------
// Exit action
	IF (me.StateMachine.intState<>me.StateMachine.intStateNext) THEN
		;
	END_IF
END_METHOD

{attribute 'object_name' := 'StateMachine'}
METHOD PROTECTED StateMachine : BOOL
SUPER^.StateMachine();

// main statemachine of base controller
CASE me.StateMachine.intState OF
	cSTA_RUNBusy: 
        THIS^.sta_RUNBusy();
	cSTA_RUN: 
        THIS^.sta_RUN();
	cSTA_MANUALBusy: 
        THIS^.sta_MANUALBusy();
	cSTA_MANUAL: 
        THIS^.sta_MANUAL();
END_CASE
END_METHOD

END_FUNCTION_BLOCK

// POUs/Controller/Lvl0/JCL (Jetter Client)/helper/cycle_Jcl
FUNCTION cycle_Jcl : BOOL
VAR_INPUT
	pJcl: POINTER TO T_JCL;
END_VAR

pJcl^.ctrl.fbJcl_Tcp();
pJcl^.ctrl.fbJcl();
pJcl^.datachn.rSendData.fbFifo();

END_FUNCTION

// POUs/Controller/Lvl0/JCL (Jetter Client)/helper/init_Jcl
FUNCTION init_Jcl : BOOL
VAR_INPUT
	pJcl: POINTER TO T_JCL;
	/// instance array of all controller instances
	pCtrlInst: POINTER TO fb_CtrlBase;
	/// common interface array of all controllers (main use for PLC)
	pCtrlCIf: POINTER TO T_Ctrl_CIf;
END_VAR

pJcl^.datachn.rSendData.fbDataChannel.InitChannel(SIZEOF(pJcl^.datachn.rSendData.rDataChannelItem), ADR(pJcl^.datachn.rSendData.rDataChannelItem));
pJcl^.datachn.rSendData.fbFifo.DataChannel := ADR(pJcl^.datachn.rSendData.fbDataChannel);
pJcl^.datachn.rSendData.fbFifo.FreeDataPointer := TRUE;
pJcl^.datachn.rSendData.fbFifo.Enable := TRUE;

pJcl^.ctrl.fbJcl_Tcp.iniAllCtrlArrays(pCtrlInst,pCtrlCIf,pJcl^.id.Jcl_Tcp);
pJcl^.ctrl.fbJcl.iniAllCtrlArrays(pCtrlInst,pCtrlCIf,pJcl^.id.Jcl);
pJcl^.ctrl.fbJcl.TCP := ADR(pJcl^.ctrl.fbJcl_Tcp);

END_FUNCTION

// POUs/Controller/Lvl0/JCL (Jetter Client)/FB_JCL
FUNCTION_BLOCK FB_JCL EXTENDS FB_CtrlBase
VAR
	/// Specific interface struct for public access
	SIf: T_Ctrl_SIf_JCL;
	/// pointer to function block
	p_fbTCP: POINTER TO FB_TCP;
	pTCP_CIF: POINTER TO BASE_PLC.T_Ctrl_CIf;
	fbStateLookup: FB_LookupTable_String;
	fbCommandLookup: FB_LookupTable;
	bolServerConnectionError: BOOL;
	/// variables for receiving msgs
	m_pDataChannel: POINTER TO FB_DataChannelSenderFifo;
END_VAR

(*__________________________________________________________________________________________________
¦	
¦	Vistaprint Schweiz GmbH
¦	CH - 8401 Winterthur
¦
¦	www.vistaprint.ch - info@vistaprint.ch
¦___________________________________________________________________________________________________

Function desription:
ToDo: DSC...

History:
Version		Date			Author				Comment
---------------------------------------------------------------------------------------------------
0.00.1		20.05.2014		AVME/DSC			Start history. Insert all basic functionalities.
___________________________________________________________________________________________________*)

SUPER^();

{attribute 'object_name' := 'Always'}
METHOD PROTECTED Always : BOOL
// not inherite from base !!!  special behaviour for this controller
// SUPER^.Always();

// Conditions Always
IF (me.bolChangeBackToAUTO=TRUE) THEN // switch mode to automatic switch off controller
	//me.StateMachine.intStateNext := cSTA_OFFBusy;
	me.bolChangeBackToAUTO := FALSE;
END_IF

IF (CIf.SwCfg.bolExist=FALSE) THEN // hardware of controller does not exist
	me.StateMachine.intStateNext := cSTA_SINGLE_ANSWER;
ELSE
	// Handle command PON
	IF (me.intCmd=cCMD_PON) 
		AND (me.StateMachine.intState<>cSTA_PONBusy) AND (me.StateMachine.intState<>cSTA_PON)
		AND (me.StateMachine.intState<>cSTA_ERROR) AND (me.StateMachine.intState<>cSTA_ERRORQuit) 
		AND (me.StateMachine.intState<>cSTA_EOFF) AND (me.StateMachine.intState<>cSTA_EOFFBusy) THEN
		me.StateMachine.intStateNext := cSTA_PONBusy;
	ELSIF (me.intCmd=cCMD_OFF) 
		AND (me.StateMachine.intState<>cSTA_PONBusy) AND (me.StateMachine.intState<>cSTA_PON)
		AND (me.StateMachine.intState<>cSTA_OFFBusy) AND (me.StateMachine.intState<>cSTA_OFF)
		AND (me.StateMachine.intState<>cSTA_ERROR) AND (me.StateMachine.intState<>cSTA_ERRORQuit) 
		AND (me.StateMachine.intState<>cSTA_EOFF) AND (me.StateMachine.intState<>cSTA_EOFFBusy)
		AND (me.StateMachine.intState<>JCL_CmdState.cSTA_MANUALMODE) THEN
		me.StateMachine.intStateNext := cSTA_OFFBusy;
	END_IF
END_IF
		
// ----------------------------------------------------------------------------------
// cyclic actions outside of statemachine
IF (me.StateMachine.intState<>cSTA_SINGLE_ANSWER) THEN
	
	// Simulation
	IF (CIf.SwCfg.bolSimulation) THEN
		;
	END_IF
	
	// Always handle recieve data from jetter server
	IF NOT CIf.SwCfg.bolSimulation THEN
		THIS^.HandleReceiveData();
	END_IF
	
	// Request state
	// ------------------------------
	IF (me.intCmd=cCMD_RequestState) THEN
		// Request state one time
		CIf.Job.intACmd := Base_PLC.cCMD_DONE;
		CIf.Job.intMCmd := Base_PLC.cCMD_DONE;
		THIS^.RequestState();
	END_IF
	
	// Reset Jetter alarms
	// ------------------------------
	// Can be done over command "cCMD_ResetAlarm" or normal global AlmReset
	IF (me.intCmd=cCMD_ResetAlarm) OR ((CIf.Job.bolAlmReset = TRUE) AND (me.StateMachine.intState<>cSTA_ERROR) AND (me.StateMachine.intState<>cSTA_ERRORQuit)) THEN
		CIf.Job.bolAlmReset := FALSE;
		IF (me.intCmd=cCMD_ResetAlarm) THEN
			CIf.Job.intACmd := Base_PLC.cCMD_DONE;
			CIf.Job.intMCmd := Base_PLC.cCMD_DONE;
		END_IF
		// Reset Jetter alarms one time
		THIS^.ResetAlarms();
	END_IF
	
	// EOFF and MANUAL
	IF (me.StateMachine.intState<>cSTA_EOFF) AND (me.StateMachine.intState<>cSTA_EOFFBusy) AND (me.StateMachine.intState>cSTA_PON)
	  AND (me.StateMachine.intState<>cSTA_ERROR) AND (me.StateMachine.intState<>cSTA_ERRORQuit)  THEN
		IF (SIf.Cur.intJETState = E_JET_STATES.EOFF) OR (SIf.Cur.intJETState = E_JET_STATES.EOFFBusy) THEN
			me.StateMachine.intStateNext := cSTA_EOFFBusy;
		ELSIF (SIf.Cur.bolIsLocalControlled) AND (me.StateMachine.intState<>cSTA_MANUALMODE) AND (me.StateMachine.intState<>cSTA_ERROR) AND (me.StateMachine.intState<>cSTA_ERRORQuit) THEN
			me.StateMachine.intStateNext := cSTA_MANUALMODE;
		END_IF
	END_IF
		
END_IF
END_METHOD

METHOD PROTECTED BarcodeArrayToUdint : UDINT
VAR_INPUT
	aBarcode 		: ARRAY[0..9] OF USINT;
END_VAR
VAR
	iIdx			: INT;
END_VAR
BarcodeArrayToUdint := 0;

FOR iIdx := 0 TO 9 DO
	BarcodeArrayToUdint := BarcodeArrayToUdint * 10 + aBarcode[iIdx];	
END_FOR
END_METHOD

{attribute 'object_name' := 'checkChildAlmClass'}
METHOD checkChildAlmClass : BOOL
// If there is a TCP connection problem to the server
IF (pTCP_CIF^.Job.eMe_ActivAlmClass >= E_AlmClass.TSTOP) THEN
	bolServerConnectionError:= TRUE;
	// set me alarm class OFF
	CIf.Job.eMe_ActivAlmClass := E_AlmClass.OFF;
	me.StateMachine.intStateNext := Base_PLC.cSTA_ERROR;
END_IF
END_METHOD

{attribute 'object_name' := 'cmdCALIBRATION'}
METHOD PROTECTED cmdCALIBRATION : BOOL
VAR
	stNextCommand: T_JCL_Command;
	pNextCommand: POINTER TO T_JCL_Command;
END_VAR
// -----------------------------------------
// Prepare telegram for CALIBRATION
// -----------------------------------------
// Define header
stNextCommand.stHeader.uinMsgId := JCL_MsgId_Command;
stNextCommand.stHeader.udiMsgSize := SIZEOF(T_JCL_Command) - SIZEOF(ST_Header);
// Set jetter CMD
stNextCommand.usiCommand := JCL_CMD_Calibration;
// Push telegram to send buffer
pNextCommand := ADR(stNextCommand);
p_fbTCP^.M_Push(paPushMsg := pNextCommand);
END_METHOD

{attribute 'object_name' := 'cmdCLEAN'}
METHOD PROTECTED cmdCLEAN : BOOL
VAR
	stNextCommand: T_JCL_Command;
	pNextCommand: POINTER TO T_JCL_Command;
END_VAR
// -----------------------------------------
// Prepare telegram for CLEAN
// -----------------------------------------
// Define header
stNextCommand.stHeader.uinMsgId := JCL_MsgId_Command;
stNextCommand.stHeader.udiMsgSize := SIZEOF(T_JCL_Command) - SIZEOF(ST_Header);
// Set jetter CMD
stNextCommand.usiCommand := JCL_CMD_CleanPrintHeads;
// Push telegram to send buffer
pNextCommand := ADR(stNextCommand);
p_fbTCP^.M_Push(paPushMsg := pNextCommand);
END_METHOD

{attribute 'object_name' := 'cmdOFF'}
METHOD PROTECTED cmdOFF : BOOL
VAR
	stNextCommand: T_JCL_Command;
	pNextCommand: POINTER TO T_JCL_Command;
END_VAR
// -----------------------------------------
// Prepare telegram for OFF
// -----------------------------------------
// Define header
stNextCommand.stHeader.uinMsgId := JCL_MsgId_Command;
stNextCommand.stHeader.udiMsgSize := SIZEOF(T_JCL_Command) - SIZEOF(ST_Header);
// Set jetter CMD
stNextCommand.usiCommand := JCL_CMD_Off;
// Push telegram to send buffer
pNextCommand := ADR(stNextCommand);
p_fbTCP^.M_Push(paPushMsg := pNextCommand);
END_METHOD

{attribute 'object_name' := 'cmdPON'}
METHOD PROTECTED cmdPON : BOOL
VAR
	stNextCommand: T_JCL_Command;
	pNextCommand: POINTER TO T_JCL_Command;
END_VAR
// -----------------------------------------
// Prepare telegram for PON
// -----------------------------------------
// Define header
stNextCommand.stHeader.uinMsgId := JCL_MsgId_Command;
stNextCommand.stHeader.udiMsgSize := SIZEOF(T_JCL_Command) - SIZEOF(ST_Header);
// Set jetter CMD
stNextCommand.usiCommand := JCL_CMD_PowerOn;
// Push telegram to send buffer
pNextCommand := ADR(stNextCommand);
p_fbTCP^.M_Push(paPushMsg := pNextCommand);
END_METHOD

{attribute 'object_name' := 'cmdRUN'}
METHOD PROTECTED cmdRUN : BOOL
VAR
	stNextCommand: T_JCL_Command;
	pNextCommand: POINTER TO T_JCL_Command;
END_VAR
// -----------------------------------------
// Prepare telegram for RUN
// -----------------------------------------
// Define header
stNextCommand.stHeader.uinMsgId := JCL_MsgId_Command;
stNextCommand.stHeader.udiMsgSize := SIZEOF(T_JCL_Command) - SIZEOF(ST_Header);
// Set jetter CMD
stNextCommand.usiCommand := JCL_CMD_Run;
// Push telegram to send buffer
pNextCommand := ADR(stNextCommand);
p_fbTCP^.M_Push(paPushMsg := pNextCommand);
END_METHOD

{attribute 'object_name' := 'cmdSTANDBY'}
METHOD PROTECTED cmdSTANDBY : BOOL
VAR
	stNextCommand: T_JCL_Command;
	pNextCommand: POINTER TO T_JCL_Command;
END_VAR
// -----------------------------------------
// Prepare telegram for STANDBY
// -----------------------------------------
// Define header
stNextCommand.stHeader.uinMsgId := JCL_MsgId_Command;
stNextCommand.stHeader.udiMsgSize := SIZEOF(T_JCL_Command) - SIZEOF(ST_Header);
// Set jetter CMD
stNextCommand.usiCommand := JCL_CMD_Standby;
// Push telegram to send buffer
pNextCommand := ADR(stNextCommand);
p_fbTCP^.M_Push(paPushMsg := pNextCommand);
END_METHOD

{attribute 'object_name' := 'CtrlInit'}
METHOD CtrlInit : BOOL
SUPER^.CtrlInit();

// one time first cyclic call!
// Open the TCP communication to jetter remote server to get the actual machine state
me.StateMachine.intStateNext := JCL_CmdState.cSTA_ConnectBusy;

// get child if
pTCP_CIF 	:= AddChild(p_fbTCP^);
END_METHOD

PROPERTY CtrlSIf : POINTER TO T_Ctrl_SIf_JCL
GET
CtrlSIf := ADR(SIf);
END_GET
END_PROPERTY

PROPERTY DataChannel : POINTER TO FB_DataChannelSenderFifo
SET
m_pDataChannel := DataChannel;
END_SET
END_PROPERTY

{attribute 'object_name' := 'FB_init'}
METHOD FB_init : BOOL
VAR_INPUT
	/// if TRUE, the retain variables are initialized (warm start / cold start)
	bInitRetains: BOOL;
	/// if TRUE, the instance afterwards gets moved into the copy code (online change)
	bInCopyCode: BOOL;
END_VAR
VAR
	iIdx: UINT;
	iLength: UINT;
END_VAR
// ------------------------------------------------------------------------------------------------------------------------
// to manually change in new FUB implementation!!!
// define valid commands for this controller
iLength := SIZEOF(CIf.Job.aCmdList)/SIZEOF(CIf.Job.aCmdList[0]);
iIdx := 0;

WHILE (iIdx < iLength) AND (CIf.Job.aCmdList[iIdx].intCmd <> cCMD_INITIALIZED) DO
	iIdx := iIdx + 1; 
END_WHILE

IF (iIdx < iLength) THEN
// Add configuration of own comands	
	CIf.Job.aCmdList[iIdx].intCmd := BASE_PLC.cCMD_RUN;
	CIf.Job.aCmdList[iIdx].strName := 'RUN'; 
	CIf.Job.aCmdList[iIdx].bolAvailable := TRUE;
    iIdx := iIdx + 1;
	CIf.Job.aCmdList[iIdx].intCmd := BASE_PLC.cCMD_STANDBY;
	CIf.Job.aCmdList[iIdx].strName := 'STANDBY'; 
	CIf.Job.aCmdList[iIdx].bolAvailable := TRUE;
	iIdx := iIdx + 1;
	CIf.Job.aCmdList[iIdx].intCmd := JCL_CmdState.cCMD_CleanPrintHeads;
	CIf.Job.aCmdList[iIdx].strName := 'CLEANING'; 
	CIf.Job.aCmdList[iIdx].bolAvailable := TRUE;
	iIdx := iIdx + 1;
	CIf.Job.aCmdList[iIdx].intCmd := JCL_CmdState.cCMD_Calibration;
	CIf.Job.aCmdList[iIdx].strName := 'CALIBRATION'; 
	CIf.Job.aCmdList[iIdx].bolAvailable := TRUE;
	iIdx := iIdx + 1;
	CIf.Job.aCmdList[iIdx].intCmd := JCL_CmdState.cCMD_ResetAlarm;
	CIf.Job.aCmdList[iIdx].strName := 'RESET ALARM'; 
	CIf.Job.aCmdList[iIdx].bolAvailable := TRUE;
	iIdx := iIdx + 1;
	CIf.Job.aCmdList[iIdx].intCmd := JCL_CmdState.cCMD_RequestState;
	CIf.Job.aCmdList[iIdx].strName := 'REQUEST STATE'; 
	CIf.Job.aCmdList[iIdx].bolAvailable := TRUE;
ELSE
	// Error if the aCmdList Array is to small
END_IF

// set name of class/typ
CIf.Info.strType := 'FB_JCL';
CIf.Info.strFullName := 'Jetter Client';

// set alarm class
SIf.Alm[E_ALM_JCL.JetterNotRun].eAlmClass := E_AlmClass.OFF;
SIf.Alm[E_ALM_JCL.JetterNotRun].strText := 'Jetter is not in RUN';
SIf.Alm[E_ALM_JCL.JetterManualWarning].eAlmClass := E_AlmClass.WARNING;
SIf.Alm[E_ALM_JCL.JetterManualWarning].strText := 'Manual Operation';
SIf.Alm[E_ALM_JCL.JetterManualError].eAlmClass := E_AlmClass.OFF;
SIf.Alm[E_ALM_JCL.JetterManualError].strText := 'Manual Operation';
SIf.Alm[E_ALM_JCL.JetterEOff].eAlmClass := E_AlmClass.OFF;
SIf.Alm[E_ALM_JCL.JetterEOff].strText := 'Jetter in EOFF';
SIf.Alm[E_ALM_JCL.JetterCommunicationLost].eAlmClass := E_AlmClass.OFF;
SIf.Alm[E_ALM_JCL.JetterCommunicationLost].strText := 'Jetter Communication Lost';
SIf.Alm[E_ALM_JCL.CleaningError].eAlmClass := E_AlmClass.OFF;
SIf.Alm[E_ALM_JCL.CleaningError].strText := 'AutoMaintenance Failed - Check Jetter';
SIf.Alm[E_ALM_JCL.DataChannelFull].eAlmClass := E_AlmClass.OFF;
SIf.Alm[E_ALM_JCL.DataChannelFull].strText := 'Print Done DataChannel Buffer is full';


// *******************************************************************************
// initial values
// *******************************************************************************

// software configuration
CIf.SwCfg.bolExist := TRUE;
CIf.SwCfg.bolEnable := TRUE;
CIf.SwCfg.bolSimulation :=  FALSE;

// Fill the lookup table with all valid jetter states
fbStateLookup.A_Add(iAddKey := E_JET_STATES.DONE			 ,strAddValue := 'DONE');
fbStateLookup.A_Add(iAddKey := E_JET_STATES.INITIALIZED		 ,strAddValue := 'INITIALIZED'	);
fbStateLookup.A_Add(iAddKey := E_JET_STATES.EOFFBusy		 ,strAddValue := 'EOFFBusy'		);
fbStateLookup.A_Add(iAddKey := E_JET_STATES.EOFF			 ,strAddValue := 'EOFF'			);
fbStateLookup.A_Add(iAddKey := E_JET_STATES.PONBusy			 ,strAddValue := 'PONbusy'		);
fbStateLookup.A_Add(iAddKey := E_JET_STATES.PON				 ,strAddValue := 'PON'			);
fbStateLookup.A_Add(iAddKey := E_JET_STATES.OFFBusy			 ,strAddValue := 'OFFbusy'		);
fbStateLookup.A_Add(iAddKey := E_JET_STATES.OFF				 ,strAddValue := 'OFF'			);
fbStateLookup.A_Add(iAddKey := E_JET_STATES.INITBusy		 ,strAddValue := 'INITbusy'		);
fbStateLookup.A_Add(iAddKey := E_JET_STATES.INIT			 ,strAddValue := 'INIT'			);
fbStateLookup.A_Add(iAddKey := E_JET_STATES.RUNBusy			 ,strAddValue := 'RUNbusy'		);
fbStateLookup.A_Add(iAddKey :=E_JET_STATES.RUN				 ,strAddValue := 'RUN'			);
fbStateLookup.A_Add(iAddKey :=E_JET_STATES.ERROR			 ,strAddValue := 'ERROR'		);
fbStateLookup.A_Add(iAddKey :=E_JET_STATES.ERRORquit		 ,strAddValue := 'ERRORquit'	);
fbStateLookup.A_Add(iAddKey :=E_JET_STATES.PARKBusy			 ,strAddValue := 'PARKbusy'		);
fbStateLookup.A_Add(iAddKey :=E_JET_STATES.PARK				 ,strAddValue := 'PARK'			);
fbStateLookup.A_Add(iAddKey :=E_JET_STATES.STANDBYBusy		 ,strAddValue := 'STANDBYbusy'	);
fbStateLookup.A_Add(iAddKey :=E_JET_STATES.STANDBY			 ,strAddValue := 'STANDBY'		);
fbStateLookup.A_Add(iAddKey :=E_JET_STATES.MAINTMANINWORK	 ,strAddValue := 'MAINTMANINWORK'	);
fbStateLookup.A_Add(iAddKey :=E_JET_STATES.MAINTMANDONE		 ,strAddValue := 'MAINTMANDONE'	);
fbStateLookup.A_Add(iAddKey :=E_JET_STATES.MAINTMANBusy		 ,strAddValue := 'MAINTMANBusy'	);
fbStateLookup.A_Add(iAddKey :=E_JET_STATES.MAINTAUTOBusy	 ,strAddValue := 'MAINTAUTOBusy'	);
fbStateLookup.A_Add(iAddKey :=E_JET_STATES.MAINTAUTODONE	 ,strAddValue := 'MAINTAUTODONE'	);
fbStateLookup.A_Add(iAddKey :=E_JET_STATES.MAINTAUTOFAILED	 ,strAddValue := 'MAINTAUTOFAILED');
fbStateLookup.A_Add(iAddKey :=E_JET_STATES.FLUSHBusy		 ,strAddValue := 'FLUSHBusy'		);
fbStateLookup.A_Add(iAddKey :=E_JET_STATES.FLUSHDONE		 ,strAddValue := 'FLUSHDONE'		);
fbStateLookup.A_Add(iAddKey :=E_JET_STATES.SPITBusy			 ,strAddValue := 'SPITBusy'		);
fbStateLookup.A_Add(iAddKey :=E_JET_STATES.SPITDONE			 ,strAddValue := 'SPITDONE'		);

SIf.Par.udiCleaningStartTimeout_ms := 5000;

SIf.Cur.bolExecuteCleaning:= FALSE;	
SIf.Cur.intJETState:= 0;  // current state not yet known
SIf.Cfg.bolJetterManualModeAllowed := FALSE;
SIf.Cfg.bolEnablePrintDoneDataChannel := FALSE;
END_METHOD

{attribute 'object_name' := 'getCmdState'}
METHOD PROTECTED getCmdState : STRING
VAR_INPUT
	intCmdState: INT;
	bolState: BOOL;
END_VAR
getCmdState := SUPER^.getCmdState(intCmdState:=intCmdState,bolState:=bolState); // get global/base defined cmds/states

IF (getCmdState='') THEN // global not defined get local
	// get string cmd/state string information in runtime	
	IF (bolState=FALSE) THEN
		// States's
		CASE intCmdState OF
			JCL_CmdState.cCMD_CleanPrintHeads: 
				getCmdState := 'CleanPrintHeads';		
				
		END_CASE;
	ELSE
		// States's
		CASE intCmdState OF			
			// Main states			
			JCL_CmdState.cSTA_ConnectBusy:
				getCmdState := 'ConnectBusy';
			JCL_CmdState.cSTA_AutoMaintenanceBusy: 
				getCmdState := 'CleanPrintHeadsBusy'; 
			JCL_CmdState.cSTA_AutoMaintenanceDone:
				getCmdState := 'CleanPrintHeads';		
			JCL_CmdState.cSTA_CalibrationBusy:
				getCmdState := 'CalibrationBusy';	
			JCL_CmdState.cSTA_Calibration:
				getCmdState := 'Calibration';	
			JCL_CmdState.cSTA_MANUALMODE:
				getCmdState := 'Jetter Manual';	
						
			// Sub states
			JCL_CmdState.cSUB_WaitingForConnection:
				getCmdState := 'WaitingForConnection';
			JCL_CmdState.cSUB_WaitingForState:
				getCmdState := 'WaitingForState';
			JCL_CmdState.cSUB_Done:
				getCmdState := 'Done';			
			JCL_CmdState.cSUB_WaitForCleaningToStart:
				getCmdState := 'WaitForCleaningToStart';
			JCL_CmdState.cSUB_CleaningBusy:
				getCmdState := 'CleaningBusy';			
		END_CASE;
	END_IF 
END_IF
END_METHOD

{attribute 'object_name' := 'getCtrlSIf'}
METHOD getCtrlSIf : POINTER TO T_Ctrl_SIf_JCL
getCtrlSIf := ADR(SIf);
END_METHOD

{attribute 'object_name' := 'HandleReceiveData'}
METHOD HandleReceiveData
VAR
	bPop			: BOOL;
	naNextMsg		: ARRAY[0..MAX_DATASET_SIZE] OF BYTE;
	pNextMsg		: POINTER TO U_JCL_Message;
END_VAR
// get next message
p_fbTCP^.M_Pop(naPopMsg => naNextMsg, bPop => bPop);
pNextMsg := ADR(naNextMsg);

IF bPop AND (pNextMsg <> NULL) THEN  // something has been recieved
	CASE pNextMsg^.State.stHeader.uinMsgId OF

		// -----------------------------------------------
		// Handle received state
		// -----------------------------------------------
		// Note: The Status is send on Request and on Status Change
		JCL_MsgId_State:
			msg_HandleState(pNextMsg);
			
		// -----------------------------------------------
		// Handle received print info (print done)
		// -----------------------------------------------		
		JCL_MsgId_PrintDone:
			msg_HandlePrintDone(pNextMsg);
		
		// -----------------------------------------------
		// Handle received alarm message
		// -----------------------------------------------
		JCL_MsgId_Alarm:
			;
			
		// -----------------------------------------------
		// Handle received request for cleaning
		// -----------------------------------------------
		JCL_MsgId_ReqCleaning:
			msg_HandleCleaningRequest(pNextMsg);	
		
		// -----------------------------------------------
		// Handle received that an automatic cleaning was done
		// -----------------------------------------------
		JCL_MsgId_CleaningDone:
			msg_HandleCleaningDone(pNextMsg);				
		
		// nothing received	
		0:
			; 
	ELSE
		; // To do: Add error	
	END_CASE
	
END_IF
END_METHOD

METHOD PROTECTED msg_HandleCleaningDone : BOOL
VAR_INPUT
	pMessage			: POINTER TO U_JCL_Message;
END_VAR
IF pMessage <> NULL THEN
	SIf.Cur.bolExecuteCleaning:= FALSE;			
	SIf.Cur.strDTOfLastCleaningCycle:= pMessage^.CleaningDone.strDTLastClean;
END_IF
END_METHOD

METHOD PROTECTED msg_HandleCleaningRequest : BOOL
VAR_INPUT
	pMessage			: POINTER TO U_JCL_Message;
END_VAR
IF pMessage <> NULL THEN
	SIf.Cur.bolExecuteCleaning:= TRUE;			
END_IF
END_METHOD

METHOD PROTECTED msg_HandlePrintDone : BOOL
VAR_INPUT
	pMessage			: POINTER TO U_JCL_Message;
END_VAR
VAR
	pItem				: POINTER TO T_JCL_DCH;
END_VAR
IF pMessage <> NULL THEN
	IF SIf.Cfg.bolEnablePrintDoneDataChannel THEN
		IF m_pDataChannel <> NULL THEN
			IF UINT_TO_INT(m_pDataChannel^.ItemCount) >= m_pDataChannel^.QueueLimit THEN
				pfbAlarmCtrl^.setAlarm(CIf.Info.intCtrlId,E_ALM_JCL.DataChannelFull,0,ADR(SIf.Alm),E_AlmState.RST,CIf.Job.eMe_ActivAlmClass);
			ELSE
				pItem := __NEW(T_JCL_DCH);
				pItem^.rBaseInfo.eHealth := E_ItemHealth.Healthy;
				pItem^.rBaseInfo.uinModuleId := 16;
				pItem^.rBaseInfo.uinActualPosition := 1;
				pItem^.udiIdentification := BarcodeArrayToUdint(pMessage^.PrintDone.usiBarcode);
				MEMCPY(ADR(pItem^.udiInkMeniscus[0]), ADR(pMessage^.PrintDone.udiInkMeniscus[0]),SIZEOF(pItem^.udiInkMeniscus)*2);
				MEMCPY(ADR(pItem^.udiPrintHeadTemperatureModule1[0]), ADR(pMessage^.PrintDone.udiPrintHeadTemperature[0,0]),SIZEOF(pItem^.udiPrintHeadTemperatureModule1[0])*5);
				MEMCPY(ADR(pItem^.udiPrintHeadTemperatureModule1[0]), ADR(pMessage^.PrintDone.udiPrintHeadTemperature[1,0]),SIZEOF(pItem^.udiPrintHeadTemperatureModule1[0])*5);
				pItem^.udiPrintLengthCalc := pMessage^.PrintDone.udiPrintLengthCalc;
				pItem^.udiPrintWidthCalc := pMessage^.PrintDone.udiPrintWidthCalc;
				pItem^.udiShiftAngleCalc := pMessage^.PrintDone.udiShiftAngleCalc;
				pItem^.udiShiftXCalc := pMessage^.PrintDone.udiShiftXCalc;
				pItem^.udiShiftYCalc := pMessage^.PrintDone.udiShiftYCalc;
				pItem^.usiInkLevelMainTank := pMessage^.PrintDone.usiInkLevelMainTank;
				pItem^.usiInkLevelReturnPrintModule1 := pMessage^.PrintDone.usiInkLevelReturnPrintModule1;
				pItem^.usiInkLevelReturnPrintModule2 := pMessage^.PrintDone.usiInkLevelReturnPrintModule2;
				pItem^.usiInkLevelSupplyPrintModule1 := pMessage^.PrintDone.usiInkLevelSupplyPrintModule1;
				pItem^.usiInkLevelSupplyPrintModule2 := pMessage^.PrintDone.usiInkLevelSupplyPrintModule2;
				m_pDataChannel^.Push(pItem);					
			END_IF
		END_IF
	END_IF
END_IF
END_METHOD

METHOD PROTECTED msg_HandleState : BOOL
VAR_INPUT
	pMessage			: POINTER TO U_JCL_Message;
END_VAR
// Update the main state
SIf.Cur.intJETState := pMessage^.State.usiMainState;
fbStateLookup.A_LookupByKey(iLookupKey := SIf.Cur.intJETState, strFoundValue => SIf.Cur.strJetState);

IF NOT fbStateLookup.bOK THEN
	SIf.Cur.strJetState := INT_TO_STRING(SIf.Cur.intJETState);
END_IF

// Prepare additional states
(*
State				   BIT		Description
-------------------------------------------------------------------------------------------------
ReadyForProduction		0		Jetter ready for production
Running					1		Print running, in production
NeedsAttention			2		System needs attention. Info or warning active
Error					3		General error active
CleaningIncomplete		4		Cleaning cycle was aborted before finishing. Production not possible.
MaintenanceInProgress	5	 	TRUE if a maintenance work is in progress. Independent if auto or manual maintenance is in progress.
IsLocalControlled		6		Local control active. Commands from Client are ignored
IsRemoteControlled		7		Remote control active. Commands from Client are accepted
CleaningRequestPending	8		Jetter requests a cleaning cylce
*)

SIf.Cur.bolReadyForProduction			:= pMessage^.State.usiAddState.0;			
SIf.Cur.bolRunning						:= pMessage^.State.usiAddState.1;		
SIf.Cur.bolNeedsAttention				:= pMessage^.State.usiAddState.2;			
SIf.Cur.bolError						:= pMessage^.State.usiAddState.3;			
SIf.Cur.bolCleaningIncomplete			:= pMessage^.State.usiAddState.4;			
SIf.Cur.bolMaintenanceInProgress		:= pMessage^.State.usiAddState.5;
SIf.Cur.bolIsLocalControlled			:= pMessage^.State.usiAddState.6;		
SIf.Cur.bolIsRemoteControlled			:= pMessage^.State.usiAddState.7;
SIf.Cur.bolCleaningRequestPending 		:= pMessage^.State.usiAddState.8;
END_METHOD

{attribute 'object_name' := 'RequestState'}
METHOD PROTECTED RequestState : BOOL
VAR
	stNextCommand: T_JCL_Command;
	pNextCommand: POINTER TO T_JCL_Command;
END_VAR
// Request jetter state
IF NOT (CIf.SwCfg.bolSimulation) THEN
	stNextCommand.stHeader.uinMsgId := JCL_MsgId_Command;
	stNextCommand.stHeader.udiMsgSize := SIZEOF(T_JCL_Command) - SIZEOF(ST_Header);
	stNextCommand.usiCommand := JCL_CMD_RequestState;
	pNextCommand := ADR(stNextCommand);	
	p_fbTCP^.M_Push(paPushMsg := pNextCommand);		
END_IF
END_METHOD

{attribute 'object_name' := 'ResetAlarms'}
METHOD PROTECTED ResetAlarms : BOOL
VAR
	stNextCommand: T_JCL_Command;
	pNextCommand: POINTER TO T_JCL_Command;
END_VAR
// Request jetter state
IF NOT (CIf.SwCfg.bolSimulation) THEN
	stNextCommand.stHeader.uinMsgId := JCL_MsgId_Command;
	stNextCommand.stHeader.udiMsgSize := SIZEOF(T_JCL_Command) - SIZEOF(ST_Header);
	stNextCommand.usiCommand := JCL_CMD_ResetAlarm;
	pNextCommand := ADR(stNextCommand);	
	p_fbTCP^.M_Push(paPushMsg := pNextCommand);		
END_IF
END_METHOD

{attribute 'object_name' := 'sta_CLEANING'}
METHOD PROTECTED sta_AUTOMAINTENANCE : BOOL
// state implemetation
// --------------------------------------------------------------------------------------
// Entry action
	IF (me.StateMachine.intState<>me.StateMachine.intStateLastCycle) THEN
		me.StateMachine.intStateLastCycle := me.StateMachine.intState;

		SIf.Cur.bolExecuteCleaning:= FALSE;			
	END_IF

// --------------------------------------------------------------------------------------
// Cyclic action
	IF (me.StateMachine.intState=me.StateMachine.intStateLastCycle) THEN
		
		CASE me.intCmd OF	
			Base_PLC.cCMD_RUN:
				me.StateMachine.intStateNext := Base_PLC.cSTA_RUNBusy;	
			BASE_PLC.cCMD_STANDBY, Base_PLC.cCMD_STOP:
				me.StateMachine.intStateNext := BASE_PLC.cSTA_STANDBYBusy;			
		END_CASE

		IF p_fbTCP^.CtrlCIf^.Job.intState <> TCP_CmdState.cSTA_Connect THEN
			pfbAlarmCtrl^.setAlarm(CIf.Info.intCtrlId,E_ALM_JCL.JetterCommunicationLost,0,ADR(SIf.Alm),E_AlmState.RST,CIf.Job.eMe_ActivAlmClass);
			me.StateMachine.intStateNext := Base_PLC.cSTA_ERROR;
		END_IF

	END_IF

// --------------------------------------------------------------------------------------
// Exit action
	IF (me.StateMachine.intState<>me.StateMachine.intStateNext) THEN
		;
	END_IF
END_METHOD

{attribute 'object_name' := 'sta_CLEANINGBusy'}
METHOD PROTECTED sta_AUTOMAINTENANCEbusy : BOOL
VAR
	stNextCommand: T_JCL_Command;
	pNextCommand: POINTER TO T_JCL_Command;
END_VAR
// state implemetation
// --------------------------------------------------------------------------------------
// Entry action
	IF (me.StateMachine.intState<>me.StateMachine.intStateLastCycle) THEN
		me.StateMachine.intStateLastCycle := me.StateMachine.intState;
		
		// Simulation
		fbSimulationTimer.IN := FALSE;
		fbSimulationTimer.PT := T#5S;
		fbSimulationTimer(); // set time/reset timer
		fbSimulationTimer.IN := TRUE; // start timer
				
		IF CIf.SwCfg.bolSimulation THEN
			;
		ELSE
			cmdCLEAN();
		END_IF

		me.SubStateMachine.intState := cSUB_WaitForCleaningToStart;		
		me.SubStateMachine.intStateNext := cSUB_WaitForCleaningToStart;		
	END_IF


// --------------------------------------------------------------------------------------
// Cyclic action
	IF (me.StateMachine.intState=me.StateMachine.intStateLastCycle) THEN
		
		// Simulation
		IF (CIf.SwCfg.bolSimulation) THEN
			fbSimulationTimer(); // simulation time
			IF (fbSimulationTimer.Q) THEN
				SIf.Cur.intJETState  := E_JET_STATES.MAINTAUTOBusy;
			END_IF
		END_IF	
		
		CASE me.SubStateMachine.intState OF
			cSUB_WaitForCleaningToStart:
				IF (SIf.Cur.intJETState = E_JET_STATES.MAINTAUTOBusy) OR (SIf.Cur.intJETState = E_JET_STATES.MAINTAUTODONE) THEN
					me.SubStateMachine.intStateNext := cSUB_CleaningBusy;
				END_IF

			cSUB_CleaningBusy:
				// Wait for feedback -> maintenance automatic done	
				IF (SIf.Cur.intJETState = E_JET_STATES.MAINTAUTODONE) AND (NOT SIf.Cur.bolCleaningRequestPending) THEN
					SIf.Cur.bolExecuteCleaning := FALSE;
					me.StateMachine.intStateNext := JCL_CmdState.cSTA_AutoMaintenanceDone;
				END_IF
		END_CASE
		
		IF SIf.Cur.intJETState = E_JET_STATES.ERROR THEN
			pfbAlarmCtrl^.setAlarm(CIf.Info.intCtrlId,E_ALM_JCL.CleaningError,0,ADR(SIf.Alm),E_AlmState.RST,CIf.Job.eMe_ActivAlmClass);
			me.SubStateMachine.intStateNext := Base_PLC.cSTA_ERROR;
		END_IF

		IF p_fbTCP^.CtrlCIf^.Job.intState <> TCP_CmdState.cSTA_Connect THEN
			pfbAlarmCtrl^.setAlarm(CIf.Info.intCtrlId,E_ALM_JCL.JetterCommunicationLost,0,ADR(SIf.Alm),E_AlmState.RST,CIf.Job.eMe_ActivAlmClass);
			me.StateMachine.intStateNext := Base_PLC.cSTA_ERROR;
		END_IF
	END_IF

// --------------------------------------------------------------------------------------
// Exit action
	IF (me.StateMachine.intState<>me.StateMachine.intStateNext) THEN
		;
	END_IF
END_METHOD

{attribute 'object_name' := 'sta_CLEANING'}
METHOD PROTECTED sta_AUTOMAINTENANCEfailed : BOOL
// state implemetation
// --------------------------------------------------------------------------------------
// Entry action
	IF (me.StateMachine.intState<>me.StateMachine.intStateLastCycle) THEN
		me.StateMachine.intStateLastCycle := me.StateMachine.intState;
		
		CIf.Job.intACmd := cCMD_DONE;
		CIf.Job.intMCmd := cCMD_DONE;

		pfbAlarmCtrl^.setAlarm(CIf.Info.intCtrlId,E_ALM_JCL.CleaningError,0,ADR(SIf.Alm),E_AlmState.RST,CIf.Job.eMe_ActivAlmClass);
		
		SIf.Cur.bolExecuteCleaning:= FALSE;			
	END_IF

// --------------------------------------------------------------------------------------
// Cyclic action
	IF (me.StateMachine.intState=me.StateMachine.intStateLastCycle) THEN
		// Only Off comand is allowed, handled in allways		

		IF p_fbTCP^.CtrlCIf^.Job.intState <> TCP_CmdState.cSTA_Connect THEN
			pfbAlarmCtrl^.setAlarm(CIf.Info.intCtrlId,E_ALM_JCL.JetterCommunicationLost,0,ADR(SIf.Alm),E_AlmState.RST,CIf.Job.eMe_ActivAlmClass);
			me.StateMachine.intStateNext := Base_PLC.cSTA_ERROR;
		END_IF

	END_IF

// --------------------------------------------------------------------------------------
// Exit action
	IF (me.StateMachine.intState<>me.StateMachine.intStateNext) THEN
		;
	END_IF
END_METHOD

{attribute 'object_name' := 'sta_CALIBRATION'}
METHOD PROTECTED sta_CALIBRATION : BOOL
// state implemetation
// --------------------------------------------------------------------------------------
// Entry action
	IF (me.StateMachine.intState<>me.StateMachine.intStateLastCycle) THEN
		me.StateMachine.intStateLastCycle := me.StateMachine.intState;
		;
	END_IF

// --------------------------------------------------------------------------------------
// Cyclic action
	IF (me.StateMachine.intState=me.StateMachine.intStateLastCycle) THEN
		
		CASE me.intCmd OF		
			BASE_PLC.cCMD_STANDBY, Base_PLC.cCMD_STOP:
				me.StateMachine.intStateNext := BASE_PLC.cSTA_STANDBYBusy;			
		END_CASE

		IF p_fbTCP^.CtrlCIf^.Job.intState <> TCP_CmdState.cSTA_Connect THEN
			pfbAlarmCtrl^.setAlarm(CIf.Info.intCtrlId,E_ALM_JCL.JetterCommunicationLost,0,ADR(SIf.Alm),E_AlmState.RST,CIf.Job.eMe_ActivAlmClass);
			me.StateMachine.intStateNext := Base_PLC.cSTA_ERROR;
		END_IF

	END_IF

// --------------------------------------------------------------------------------------
// Exit action
	IF (me.StateMachine.intState<>me.StateMachine.intStateNext) THEN
		;
	END_IF
END_METHOD

{attribute 'object_name' := 'sta_CALIBRATIONBusy'}
METHOD PROTECTED sta_CALIBRATIONBusy : BOOL
VAR
	stNextCommand: T_JCL_Command;
	pNextCommand: POINTER TO T_JCL_Command;
END_VAR
// state implemetation
// --------------------------------------------------------------------------------------
// Entry action
	IF (me.StateMachine.intState<>me.StateMachine.intStateLastCycle) THEN
		me.StateMachine.intStateLastCycle := me.StateMachine.intState;
		
		// Simulation
		fbSimulationTimer.IN := FALSE;
		fbSimulationTimer.PT := T#5S;
		fbSimulationTimer(); // set time/reset timer
		fbSimulationTimer.IN := TRUE; // start timer
				
		IF CIf.SwCfg.bolSimulation THEN
			;
		ELSE
			cmdCALIBRATION();
		END_IF
		
	END_IF

// --------------------------------------------------------------------------------------
// Cyclic action
	IF (me.StateMachine.intState=me.StateMachine.intStateLastCycle) THEN
		
		// Simulation
		IF (CIf.SwCfg.bolSimulation) THEN
			fbSimulationTimer(); // simulation time
			IF (fbSimulationTimer.Q) THEN
				SIf.Cur.intJETState  := E_JET_STATES.CALIBRATE;
			END_IF
		END_IF	
	
		// Wait for feedback -> maintenance automatic done	
		IF (SIf.Cur.intJETState = E_JET_STATES.CALIBRATE) THEN
			me.StateMachine.intStateNext := JCL_CmdState.cSTA_Calibration;
		END_IF
		
		IF p_fbTCP^.CtrlCIf^.Job.intState <> TCP_CmdState.cSTA_Connect THEN
			pfbAlarmCtrl^.setAlarm(CIf.Info.intCtrlId,E_ALM_JCL.JetterCommunicationLost,0,ADR(SIf.Alm),E_AlmState.RST,CIf.Job.eMe_ActivAlmClass);
			me.StateMachine.intStateNext := Base_PLC.cSTA_ERROR;
		END_IF

		
	END_IF

// --------------------------------------------------------------------------------------
// Exit action
	IF (me.StateMachine.intState<>me.StateMachine.intStateNext) THEN
		;
	END_IF
END_METHOD

{attribute 'object_name' := 'sta_CONNECTBusy'}
METHOD sta_CONNECTBusy : BOOL
VAR
	stNextCommand: T_JCL_Command;
	pNextCommand: POINTER TO T_JCL_Command;
END_VAR
// state implemetation
// --------------------------------------------------------------------------------------
// Entry action
	IF (me.StateMachine.intState<>me.StateMachine.intStateLastCycle) THEN
		me.StateMachine.intStateLastCycle := me.StateMachine.intState;
	
		// **********************************************************************************
		// This state will be executed one time after startup or after an error ack.
		// State open the TCP communication to jetter remote server to get the actual machine state
		// **********************************************************************************
		// Reset state 
		SIf.Cur.intJETState:= 0;
		
		// Connect to the jetter server
		pTCP_CIF^.Job.intACmd:= TCP_CmdState.cCMD_Connect;
		
		// Initialize sub state machine
		me.SubStateMachine.intStateNext:= JCL_CmdState.cSUB_WaitingForConnection;		
		me.SubStateMachine.intState:= me.SubStateMachine.intStateNext-1;
	END_IF

// --------------------------------------------------------------------------------------
// Cyclic action
	IF (me.StateMachine.intState=me.StateMachine.intStateLastCycle) THEN
		
		// -----------------------------------------------
		// Sub state machine handle 
		// -----------------------------------------------
		CASE me.SubStateMachine.intState OF
			
			JCL_CmdState.cSUB_WaitingForConnection:			
				// Wait for connection
				IF (pTCP_CIF^.Job.intState = TCP_CmdState.cSTA_Connect) THEN	
					// Request jetter states the first time after TCP client connected				
					THIS^.RequestState();		
					me.SubStateMachine.intStateNext:= JCL_CmdState.cSUB_WaitingForState;	
				END_IF
			
			JCL_CmdState.cSUB_WaitingForState:
				// Wait for first status msg 
				IF (SIf.Cur.intJETState > 0) THEN 
					me.SubStateMachine.intStateNext:= JCL_CmdState.cSUB_Done;
				END_IF	

			JCL_CmdState.cSUB_Done:
				// Change to the init state
				me.StateMachine.intStateNext := SIf.Cur.intJETState;
			
		END_CASE
			
	END_IF

// --------------------------------------------------------------------------------------
// Exit action
	IF (me.StateMachine.intState<>me.StateMachine.intStateNext) THEN
		;
	END_IF
END_METHOD

